Omron CX-Programmer project WWFH320 (CX-Programmer 9.73)

# PLC CPM2A: CPM2* 

## Global symbols (name address type ; comment)
0.00 BOOL  ; $?St$Bk?_#[4] / LS1 AREA SENSOR / $?St$Bk?_#[4]
0.01 BOOL  ; LS2 index origin
0.02 BOOL  ; LS3A WORK DETECT
0.03 BOOL  ; LS3B WORK DETECT
0.04 BOOL  ; LS4A WORK DETECT
0.05 BOOL  ; LS4B WORK DETECT
0.06 BOOL  ; LS5A WORK DETECT
0.07 BOOL  ; LS5B WORK DETECT
0.08 BOOL  ; LS6A WORK DETECT
0.09 BOOL  ; LS6B WORK DETECT
10.00 BOOL  ; SSR1 index start
10.01 BOOL  ; $?St$Bk?_#[5] / SSR2 INDEX CW / �$?St$Bk?_#[5]
10.02 BOOL  ; $?St$Bk?_#[6] / SSR3 INDEX CCW / $?St$Bk?_#[6]
10.03 BOOL  ; SSR4 OK SIGNAL T
10.04 BOOL  ; SOL1 ROTALY TABL
10.05 BOOL  ; shower flow on
10.06 BOOL  ; SOL3 air blow on
11.01 BOOL  ; M2,M4 ON
11.02 BOOL  ; MS5 work rotatio
11.06 BOOL  ; PL5A CYCLE RUN(G
11.07 BOOL  ; PL5B CYCLE RUN(R
12 CHANNEL  ; 7seg out channel
12.04 BOOL  ; 7SEG BLANK
12.05 BOOL  ; PL3 HOME POSITIO
12.06 BOOL  ; $?St$Bk?_#[7] / PL4 ALARM / 堎忢$?St$Bk?_#[7]
12.07 BOOL  ; $?St$Bk?_#[8] / PUMP MOTOR ON / �$?St$Bk?_#[8]
18.00 BOOL  ; cycle time displ
18.01 BOOL  ; cycle time displ
18.02 BOOL  ; cycle time displ
1.00 BOOL  ; PS1 AIR PRESSURE
1.01 BOOL  ; $?St$Bk?_#[9] / WORK OK SIGNAL / $?St$Bk?_#[9]
1.02 BOOL  ; MS0 CONTROL POWE
1.03 BOOL  ; CP1 INDEX PROTEC
1.06 BOOL  ; TS1 CYCLE START
1.07 BOOL  ; PB5 2HAND丂INTER
1.08 BOOL  ; PB8 PUMP MOTOR O
1.09 BOOL  ; PB9 PUMP MOTOR O
1.10 BOOL  ; PB3 ORIGIN丂CHEC
1.11 BOOL  ; $?St$Bk?_#[10] / PB4 alarm reset / $?St$Bk?_#[10]
200.00 BOOL  ; $?St$Bk?_#[11] / WORK OK / 馨窸K$?St$Bk?_#[11]
20.00 BOOL  ; $?St$Bk?_#[12] / CYCLE HAND ON / �$?St$Bk?_#[12]
20.01 BOOL  ; $?St$Bk?_#[13] / CYCLE HAND OFF / $?St$Bk?_#[13]
20.02 BOOL  ; $?St$Bk?_#[14] / INDEX RIGHT / 草�$?St$Bk?_#[14]
20.04 BOOL  ; $?St$Bk?_#[15] / INDEX LEFT / 草棉$?St$Bk?_#[15]
20.06 BOOL  ; WORK ROTATION ON
20.07 BOOL  ; WORK ROTATION OF
20.08 BOOL  ; ROTALT TABLE DOW
20.09 BOOL  ; $?St$Bk?_#[16] / rotary table up / $?St$Bk?_#[16]
20.10 BOOL  ; $?St$Bk?_#[17] / SHOWER ON / 愻忩$?St$Bk?_#[17]
20.11 BOOL  ; $?St$Bk?_#[18] / SHOWER OFF / 愻忩$?St$Bk?_#[18]
20.12 BOOL  ; $?St$Bk?_#[19] / AIR BLOW ON / 幢�$?St$Bk?_#[19]
20.13 BOOL  ; $?St$Bk?_#[20] / AIR BLOW OFF / 幢$?St$Bk?_#[20]
210.00 BOOL  ; $?St$Bk?_#[21] / ALARM CODE SET / $?St$Bk?_#[21]
211.14 BOOL  ; ALARM CODE SHIFT
212.00 BOOL  ; $?St$Bk?_#[22] / ALARM CODE ON / �$?St$Bk?_#[22]
212.01 BOOL  ; $?St$Bk?_#[23] / NEXT NG CODE / 師$?St$Bk?_#[23]
212.02 BOOL  ; NEXT ALARM CODE
212.04 BOOL  ; ALARM CODE CLEAR
213.01 BOOL  ; $?St$Bk?_#[25] / ALARM CODE "B" / $?St$Bk?_#[25]
213.02 BOOL  ; $?St$Bk?_#[26] / ALARM CODE "C" / $?St$Bk?_#[26]
213.03 BOOL  ; $?St$Bk?_#[27] / ALARM CODE "D" / $?St$Bk?_#[27]
220.00 BOOL  ; $?St$Bk?_#[28] / ALARM CODE OFF / $?St$Bk?_#[28]
23.00 BOOL  ; CONTROL POWER ON
23.01 BOOL  ; TS1 CYCLE START
23.02 BOOL  ; $?St$Bk?_#[29] / ORIGIN CHECK / 尨$?St$Bk?_#[29]
23.03 BOOL  ; $?St$Bk?_#[30] / ALARM RESET / 堎$?St$Bk?_#[30]
24.00 BOOL  ; $?St$Bk?_#[31] / INDEX ENABLE / 草$?St$Bk?_#[31]
253.08 BOOL  ; CPU BATTERY DOWN
253.10 BOOL  ; CPU I/O UNIT ERR
25.00 BOOL  ; HAND MODE丂INABL
26.00 BOOL  ; $?St$Bk?_#[32] / INDEX RIGHT / 草�$?St$Bk?_#[32]
26.02 BOOL  ; $?St$Bk?_#[33] / INDEX LEFT / 草棉$?St$Bk?_#[33]
26.04 BOOL  ; $?St$Bk?_#[34] / INDEX RIGHT / 草�$?St$Bk?_#[34]
26.06 BOOL  ; $?St$Bk?_#[35] / INDEX RIGHT / 草�$?St$Bk?_#[35]
26.08 BOOL  ; $?St$Bk?_#[36] / INDEX RIGHT END / $?St$Bk?_#[36]
26.10 BOOL  ; $?St$Bk?_#[37] / INDEX LEFT / 草棉$?St$Bk?_#[37]
26.12 BOOL  ; $?St$Bk?_#[38] / INDEX LEFT / 草棉$?St$Bk?_#[38]
26.14 BOOL  ; $?St$Bk?_#[39] / INDEX LEFT END / $?St$Bk?_#[39]
27.00 BOOL  ; WORK ROTATION ON
27.02 BOOL  ; WORK ROTATION OF
27.06 BOOL  ; $?St$Bk?_#[40] / SHOWER ON / 愻忩$?St$Bk?_#[40]
27.08 BOOL  ; $?St$Bk?_#[41] / SHOWER OFF / 愻忩$?St$Bk?_#[41]
27.10 BOOL  ; $?St$Bk?_#[42] / SHOWER ON / 愻忩$?St$Bk?_#[42]
27.12 BOOL  ; rotary table dow
27.14 BOOL  ; $?St$Bk?_#[43] / rotary table up / $?St$Bk?_#[43]
28.00 BOOL  ; $?St$Bk?_#[44] / AIR BLOW ON / 幢�$?St$Bk?_#[44]
28.02 BOOL  ; $?St$Bk?_#[45] / AIR BLOW OFF / 幢$?St$Bk?_#[45]
29.00 BOOL  ; $?St$Bk?_#[46] / PUMP MOTOR ON / �$?St$Bk?_#[46]
2.00 BOOL  ; $?St$Bk?_#[47] / SS1 CYCLE HAND / $?St$Bk?_#[47]
2.01 BOOL  ; $?St$Bk?_#[48] / SS2 INDEX RIGHT / $?St$Bk?_#[48]
2.02 BOOL  ; $?St$Bk?_#[49] / SS2 INDEX LEFT / $?St$Bk?_#[49]
2.03 BOOL  ; SS3 WORK ROTATIO
2.04 BOOL  ; SS4 ROTALT TABLE
2.05 BOOL  ; $?St$Bk?_#[50] / SS5 SHOWER ON / $?St$Bk?_#[50]
2.06 BOOL  ; $?St$Bk?_#[51] / SS6 AIR BLOW ON / $?St$Bk?_#[51]
2.07 BOOL  ; SW1 WORK DETECT
2.08 BOOL  ; WASHER FLOW SWIT
2.10 BOOL  ; FS2 WASHER LIQUI
30.00 BOOL  ; return cycle run
30.01 BOOL  ; return cycle 1cm
30.02 BOOL  ; return cycle 2cm
30.13 BOOL  ; return cycle ind
30.14 BOOL  ; return cycle ind
30.15 BOOL  ; return complete
31.00 BOOL  ; WORK DETECT IN 1
31.01 BOOL  ; WORK DETECT IN 2
31.02 BOOL  ; NO WORK DETECT I
31.03 BOOL  ; $?St$Bk?_#[52] / WORK DETECT OUT / $?St$Bk?_#[52]
31.04 BOOL  ; NO WORK DETECT O
31.05 BOOL  ; WORK DETECT IN丂
31.06 BOOL  ; WORK DETECT IN俀
32.00 BOOL  ; $?St$Bk?_#[53] / HAND MODE / 庤摦�$?St$Bk?_#[53]
32.01 BOOL  ; $?St$Bk?_#[54] / CYCLE AUTO / 帺摦$?St$Bk?_#[54]
32.05 BOOL  ; work OK signal c
32.09 BOOL  ; $?St$Bk?_#[55] / MAIN AIR OK / 嬻$?St$Bk?_#[55]
32.10 BOOL  ; $?St$Bk?_#[56] / SWITCH OK / AUTO$?St$Bk?_#[56]
32.11 BOOL  ; $?St$Bk?_#[57] / SWITCH OK / 讲�罯$?St$Bk?_#[57]
32.12 BOOL  ; $?St$Bk?_#[58] / LS OK / 匦�慕帛罯$?St$Bk?_#[58]
32.13 BOOL  ; $?St$Bk?_#[59] / SOL OK / 口刹霓OK$?St$Bk?_#[59]
32.14 BOOL  ; INDEX PROTECTOR
32.15 BOOL  ; $?St$Bk?_#[60] / MACHIN ORIGIN / $?St$Bk?_#[60]
33.00 BOOL  ; $?St$Bk?_#[61] / EMERGENCY STOP / $?St$Bk?_#[61]
33.02 BOOL  ; $?St$Bk?_#[62] / CYCLE STOP / 徊纲$?St$Bk?_#[62]
33.15 BOOL  ; $?St$Bk?_#[63] / HOME POSITION / $?St$Bk?_#[63]
34.00 BOOL  ; $?St$Bk?_#[64] / CYCLE RUN / 婲摦$?St$Bk?_#[64]
34.01 BOOL  ; $?St$Bk?_#[65] / CYCLE START / 徊�$?St$Bk?_#[65]
34.02 BOOL  ; cycle stat comma
34.03 BOOL  ; CYCLE MEMORY CLE
34.04 BOOL  ; work=1丄馨�1屄棳
34.05 BOOL  ; 楢懕徊纲
34.06 BOOL  ; $?St$Bk?_#[66] / AUTO CYCLE OFF / $?St$Bk?_#[66]
3.00 BOOL  ; LS7 rotary table
3.01 BOOL  ; LS8 ROTARY TABLE
3.02 BOOL  ; THR1 CLEAN TANK
3.06 BOOL  ; OL2 WASHER PUMP
3.08 BOOL  ; OL4 MISTPURE MOT
3.09 BOOL  ; OL5 WORK ROTATIO
3.10 BOOL  ; M2 M4 ON
40.00 BOOL  ; index right comm
40.02 BOOL  ; index right turn
40.04 BOOL  ; iindex right fin
40.06 BOOL  ; rotary table not
41.00 BOOL  ; rotary table dow
41.01 BOOL  ; rotary table dow
41.02 BOOL  ; work rotation mo
41.03 BOOL  ; $?St$Bk?_#[67] / shower flow fin / $?St$Bk?_#[67]
41.04 BOOL  ; air brow command
41.05 BOOL  ; $?St$Bk?_#[68] / air brow fin / 幢$?St$Bk?_#[68]
41.06 BOOL  ; work丂rotaition
41.07 BOOL  ; work丂rotaition
41.08 BOOL  ; rotary table up
41.09 BOOL  ; rotary table up
42.00 BOOL  ; $?St$Bk?_#[69] / first cycle end / $?St$Bk?_#[69]
42.01 BOOL  ; $?St$Bk?_#[70] / 2nd cycle end / $?St$Bk?_#[70]
42.02 BOOL  ; 2nd cycle start
42.04 BOOL  ; $?St$Bk?_#[71] / 2nd cycle end / $?St$Bk?_#[71]
47.00 BOOL  ; $?St$Bk?_#[72] / index right / 草�$?St$Bk?_#[72]
47.02 BOOL  ; index right turn
47.04 BOOL  ; $?St$Bk?_#[73] / index right end / $?St$Bk?_#[73]
49.00 BOOL  ; $?St$Bk?_#[74] / cycle Ffinish / $?St$Bk?_#[74]
DM0 CHANNEL  ; PROGRAM VERSION
DM1 CHANNEL  ; CYCLE TIME COUNT
DM10 CHANNEL  ; $?St$Bk?_#[75] / CYCLE COUNT / 徊�$?St$Bk?_#[75]
DM120 CHANNEL  ; shower flow time
DM121 CHANNEL  ; $?St$Bk?_#[76] / air blow timer / $?St$Bk?_#[76]
DM2 CHANNEL  ; CYCLE TIME
HR10.00 BOOL  ; AIR PRESSURE ALA
HR10.02 BOOL  ; WASHER PUMP MOTO
HR10.03 BOOL  ; 丂
HR10.04 BOOL  ; MISTPURE MOTOR O
HR10.05 BOOL  ; WORK ROTATION  M
HR10.06 BOOL  ; $?St$Bk?_#[77] / AREA SENSOR OFF / $?St$Bk?_#[77]
HR10.07 BOOL  ; NDEX PROTECTOR N
HR10.08 BOOL  ; CONTROL POWER OF
HR10.09 BOOL  ; $?St$Bk?_#[78] / PLC丂ALARM / 及馆$?St$Bk?_#[78]
HR11.00 BOOL  ; INDEX TIME OVER
HR11.01 BOOL  ; ROTALY TABLE UP/
HR11.03 BOOL  ; M2,M4 ALARM
HR11.04 BOOL  ; WASHER FLOW SWIT
HR11.08 BOOL  ; $?St$Bk?_#[79] / INDEX WORK NG / �$?St$Bk?_#[79]
HR11.09 BOOL  ; $?St$Bk?_#[80] / CYCLE TIME OVER / $?St$Bk?_#[80]
HR11.15 BOOL  ; return cycle tim
HR12.00 BOOL  ; $?St$Bk?_#[81] / LS POSITION NG / $?St$Bk?_#[81]
HR12.01 BOOL  ; SWITCH POSITION
HR12.02 BOOL  ; IOK SIGNAL NOT C
HR12.04 BOOL  ; WORK DETECT IN N
HR12.05 BOOL  ; WORK DETECT OUT
HR12.06 BOOL  ; $?St$Bk?_#[82] / SOL NG / 口刹霓尨$?St$Bk?_#[82]
HR13.00 BOOL  ; SWITCH POSITION
HR13.02 BOOL  ; CLEAN TANK TEMP
HR13.03 BOOL  ; $?St$Bk?_#[83] / WASHER LEVEL NG / $?St$Bk?_#[83]
HR14.00 BOOL  ; EMERGENCY STOP A
HR14.01 BOOL  ; EMERGENCY STOP A
HR14.02 BOOL  ; EMERGENCY STOP A
HR14.03 BOOL  ; CYCLE STOP ALARM
HR14.10 BOOL  ; $?St$Bk?_#[84] / ALARM / 憤崌堎忢$?St$Bk?_#[84]
HR14.11 BOOL  ; $?St$Bk?_#[85] / ALARM ON / 弊把敪$?St$Bk?_#[85]
HR19.00 BOOL  ; 嫙媼晹馨妇莼皸L
TIM000 BOOL  ; CYCLE TIME OVER
TIM002 BOOL  ; 2HAND INTERLOCK
TIM005 BOOL  ; $?St$Bk?_#[86] / alarm reset ON / $?St$Bk?_#[86]
TIM009 BOOL  ; rotary table dow
TIM010 BOOL  ; $?St$Bk?_#[87] / INDEX RIGTH END / $?St$Bk?_#[87]
TIM011 BOOL  ; shower flow time
TIM012 BOOL  ; $?St$Bk?_#[88] / air blow timer / $?St$Bk?_#[88]
TIM013 BOOL  ; work丂rotation m
TIM020 BOOL  ; INDEX TIME OVER
TIM021 BOOL  ; ROTALY TABLE UP/
TIM023 BOOL  ; M2,M4 ALARM
TIM025 BOOL  ; WASHER FLOW SWIT
TIM029 BOOL  ; 楢懕徊纲婲摦
TIM030 BOOL  ; SOL2 shower flow
TIM031 BOOL  ; SOL2 shower flow
TIM050 BOOL  ; ALARM CODE A TO
TIM051 BOOL  ; ALARM CODE 0 TO
TIM052 BOOL  ; NEXT ALARM CODE
TIM130 BOOL  ; return start che
TIM131 BOOL  ; return cycle tim
TIM133 BOOL  ; return cycle com

## Program 怴婯踢鄹拮�1 (no task)

### Section VERSION
; 这套PLC程序设计用于控制一台轴承自动检测机，与上位机NT31-ST123协同工作。 / 程序实现了手动和自动两种操作模式。 / 将PLC控制器，连接循环手动开关、索引开关、工件旋转开关、旋转台开关、喷淋开关、气吹开关、双手互锁按钮、工件检测传感器、原点位置传感器、气压检测传感器、清洗泵、气吹装置、报警灯、7段显示器等设备。 / 在手动模式下，操作员通过按下循环手动开关切换模式，置位手动模式使能，即可通过索引右开关和索引左开关控制索引启动继电器的方向，调整轴承位置。按下工件旋转开关触发工件旋转电机控制继电器，使工件旋转以便检查。通过旋转台开关操作旋转台控制电磁阀升降旋转台，但下降时需双手互锁开关置位以保障安全。按下喷淋开关开启喷淋控制电磁阀进行清洗，或按下气吹开关启动气吹控制电磁阀吹干水分。手动操作通过7段显示输出通道实时展示状态。 / 在自动模式下，操作员按下循环启动按钮触发流程，系统检查原点位置标志是否置位，只有设备处于原点位置时循环运行标志才会置位并开始运行，同时需确保工件检测传感器A和工件检测传感器B置位以确认工件到位。若双手互锁置位且循环启动触发，系统进入自动模式准备状态。当循环启动命令置位后，系统记录工件检测状态以备后续检查。若工件检测B与开关同时置位，确认工件到位信号。自动流程按顺序执行：索引启动继电器将轴承移至检测位，旋转台控制电磁阀下降至清洗位，工件旋转电机控制继电器启动以均匀清洗轴承表面。接着，喷淋控制电磁阀开启进行清洗，此时需工件检测传感器A置位以确认工件存在。随后，气吹控制电磁阀吹干水分，需旋转台下降传感器置位以保证旋转台在下降位。当旋转台下降传感器置位时，确认旋转台下降到位信号。清洗吹干完成后，旋转台控制电磁阀上升复位，循环计数存储记录检测次数，最终通过OK信号继电器输出检测结果。 / 运行过程中，系统通过7段显示输出通道显示状态。若气压检测传感器检测到气压低于阈值或清洗泵过载传感器置位，循环运行标志立即复位，报警指示灯亮起，7段显示输出通道显示报警代码，系统进入紧急停止标志状态。操作员按下报警复位按钮后，只有当所有异常条件清除时，报警指示灯才会熄灭，系统恢复运行。

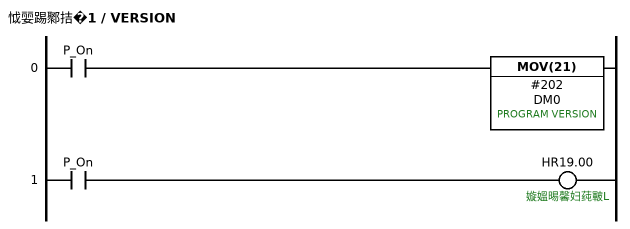
; rung 0
LD P_On
MOV(21) #202 DM0  ; PROGRAM VERSION
; rung 1
LD P_On
OUT HR19.00  ; 嫙媼晹馨妇莼皸L

### Section CYCLE_SET

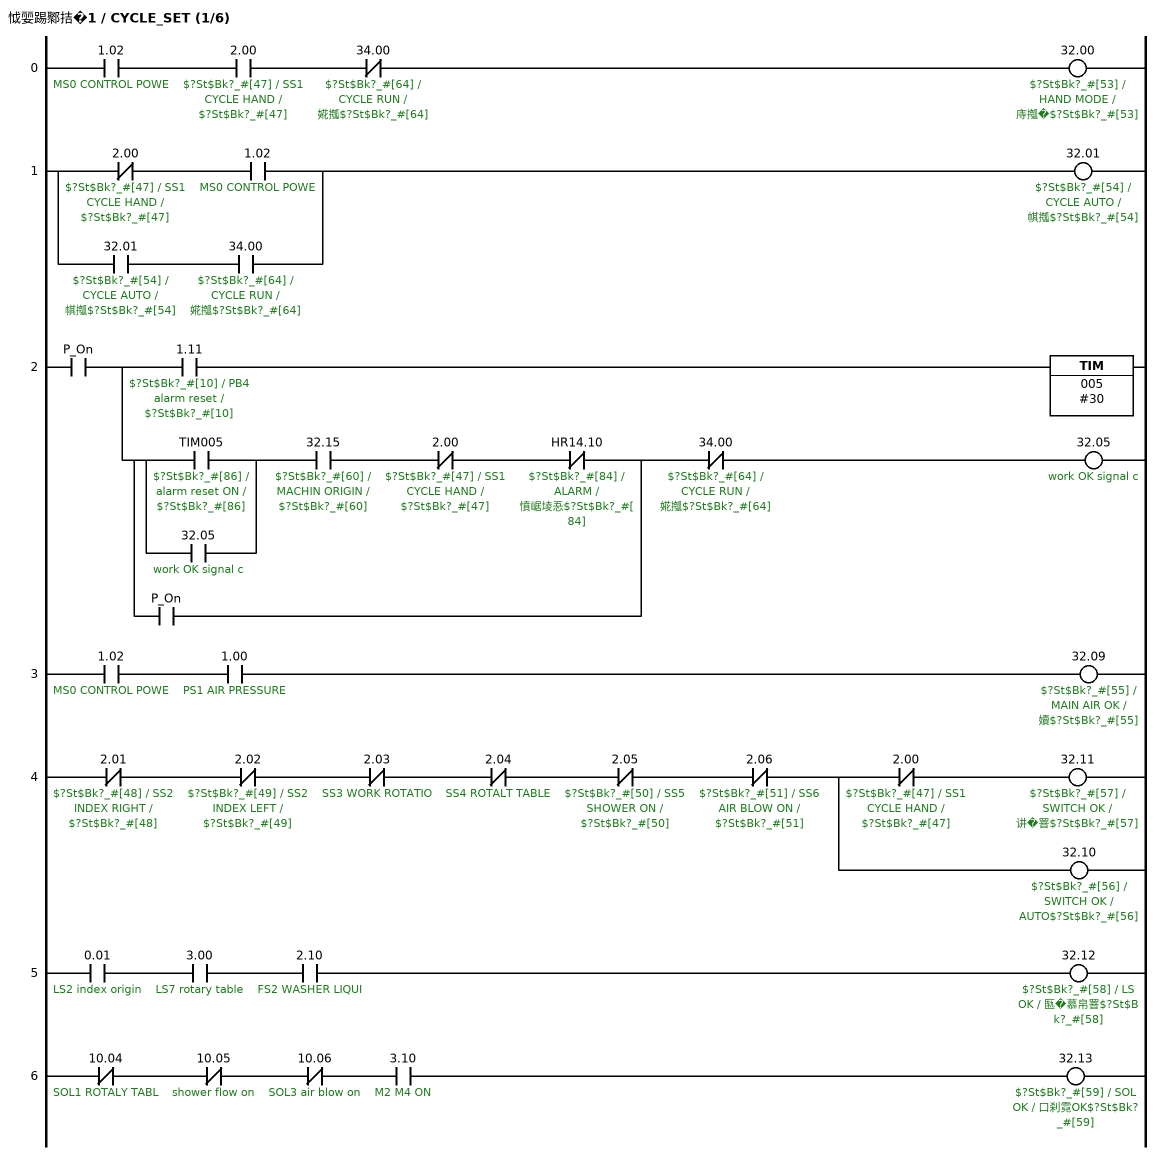
; rung 0
LD 1.02  ; MS0 CONTROL POWE
AND 2.00  ; $?St$Bk?_#[47] / SS1 CYCLE HAND / $?St$Bk?_#[47]
ANDNOT 34.00  ; $?St$Bk?_#[64] / CYCLE RUN / 婲摦$?St$Bk?_#[64]
OUT 32.00  ; $?St$Bk?_#[53] / HAND MODE / 庤摦�$?St$Bk?_#[53]
; rung 1
LDNOT 2.00  ; $?St$Bk?_#[47] / SS1 CYCLE HAND / $?St$Bk?_#[47]
AND 1.02  ; MS0 CONTROL POWE
LD 32.01  ; $?St$Bk?_#[54] / CYCLE AUTO / 帺摦$?St$Bk?_#[54]
AND 34.00  ; $?St$Bk?_#[64] / CYCLE RUN / 婲摦$?St$Bk?_#[64]
ORLD
OUT 32.01  ; $?St$Bk?_#[54] / CYCLE AUTO / 帺摦$?St$Bk?_#[54]
; rung 2
LD P_On
OUT TR0
AND 1.11  ; $?St$Bk?_#[10] / PB4 alarm reset / $?St$Bk?_#[10]
TIM 005 #30
LD TR0
LD TIM005  ; $?St$Bk?_#[86] / alarm reset ON / $?St$Bk?_#[86]
OR 32.05  ; work OK signal c
AND 32.15  ; $?St$Bk?_#[60] / MACHIN ORIGIN / $?St$Bk?_#[60]
ANDNOT 2.00  ; $?St$Bk?_#[47] / SS1 CYCLE HAND / $?St$Bk?_#[47]
ANDNOT HR14.10  ; $?St$Bk?_#[84] / ALARM / 憤崌堎忢$?St$Bk?_#[84]
OR P_On
ANDLD
ANDNOT 34.00  ; $?St$Bk?_#[64] / CYCLE RUN / 婲摦$?St$Bk?_#[64]
OUT 32.05  ; work OK signal c
; rung 3
LD 1.02  ; MS0 CONTROL POWE
AND 1.00  ; PS1 AIR PRESSURE
OUT 32.09  ; $?St$Bk?_#[55] / MAIN AIR OK / 嬻$?St$Bk?_#[55]
; rung 4
LDNOT 2.01  ; $?St$Bk?_#[48] / SS2 INDEX RIGHT / $?St$Bk?_#[48]
ANDNOT 2.02  ; $?St$Bk?_#[49] / SS2 INDEX LEFT / $?St$Bk?_#[49]
ANDNOT 2.03  ; SS3 WORK ROTATIO
ANDNOT 2.04  ; SS4 ROTALT TABLE
ANDNOT 2.05  ; $?St$Bk?_#[50] / SS5 SHOWER ON / $?St$Bk?_#[50]
ANDNOT 2.06  ; $?St$Bk?_#[51] / SS6 AIR BLOW ON / $?St$Bk?_#[51]
OUT TR0
ANDNOT 2.00  ; $?St$Bk?_#[47] / SS1 CYCLE HAND / $?St$Bk?_#[47]
OUT 32.11  ; $?St$Bk?_#[57] / SWITCH OK / 讲�罯$?St$Bk?_#[57]
LD TR0
OUT 32.10  ; $?St$Bk?_#[56] / SWITCH OK / AUTO$?St$Bk?_#[56]
; rung 5
LD 0.01  ; LS2 index origin
AND 3.00  ; LS7 rotary table
AND 2.10  ; FS2 WASHER LIQUI
OUT 32.12  ; $?St$Bk?_#[58] / LS OK / 匦�慕帛罯$?St$Bk?_#[58]
; rung 6
LDNOT 10.04  ; SOL1 ROTALY TABL
ANDNOT 10.05  ; shower flow on
ANDNOT 10.06  ; SOL3 air blow on
AND 3.10  ; M2 M4 ON
OUT 32.13  ; $?St$Bk?_#[59] / SOL OK / 口刹霓OK$?St$Bk?_#[59]

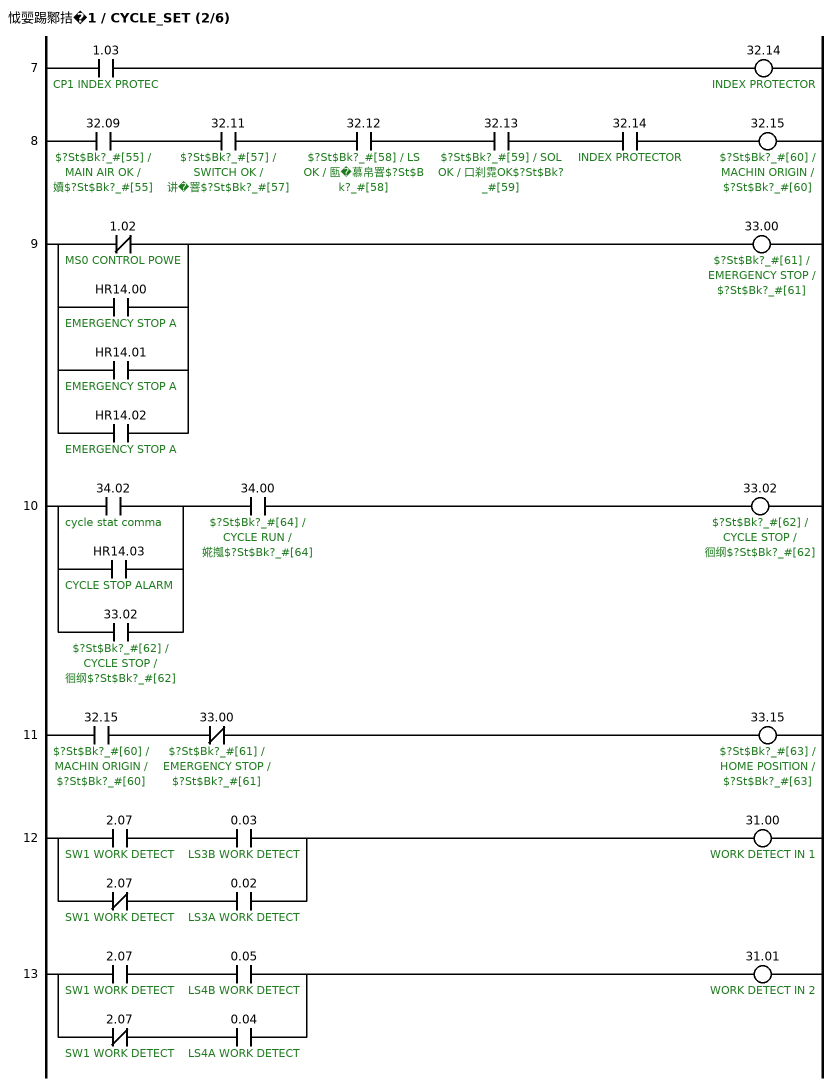
; rung 7
LD 1.03  ; CP1 INDEX PROTEC
OUT 32.14  ; INDEX PROTECTOR
; rung 8
LD 32.09  ; $?St$Bk?_#[55] / MAIN AIR OK / 嬻$?St$Bk?_#[55]
AND 32.11  ; $?St$Bk?_#[57] / SWITCH OK / 讲�罯$?St$Bk?_#[57]
AND 32.12  ; $?St$Bk?_#[58] / LS OK / 匦�慕帛罯$?St$Bk?_#[58]
AND 32.13  ; $?St$Bk?_#[59] / SOL OK / 口刹霓OK$?St$Bk?_#[59]
AND 32.14  ; INDEX PROTECTOR
OUT 32.15  ; $?St$Bk?_#[60] / MACHIN ORIGIN / $?St$Bk?_#[60]
; rung 9
LDNOT 1.02  ; MS0 CONTROL POWE
OR HR14.00  ; EMERGENCY STOP A
OR HR14.01  ; EMERGENCY STOP A
OR HR14.02  ; EMERGENCY STOP A
OUT 33.00  ; $?St$Bk?_#[61] / EMERGENCY STOP / $?St$Bk?_#[61]
; rung 10
LD 34.02  ; cycle stat comma
OR HR14.03  ; CYCLE STOP ALARM
OR 33.02  ; $?St$Bk?_#[62] / CYCLE STOP / 徊纲$?St$Bk?_#[62]
AND 34.00  ; $?St$Bk?_#[64] / CYCLE RUN / 婲摦$?St$Bk?_#[64]
OUT 33.02  ; $?St$Bk?_#[62] / CYCLE STOP / 徊纲$?St$Bk?_#[62]
; rung 11
LD 32.15  ; $?St$Bk?_#[60] / MACHIN ORIGIN / $?St$Bk?_#[60]
ANDNOT 33.00  ; $?St$Bk?_#[61] / EMERGENCY STOP / $?St$Bk?_#[61]
OUT 33.15  ; $?St$Bk?_#[63] / HOME POSITION / $?St$Bk?_#[63]
; rung 12
LD 2.07  ; SW1 WORK DETECT
AND 0.03  ; LS3B WORK DETECT
LDNOT 2.07  ; SW1 WORK DETECT
AND 0.02  ; LS3A WORK DETECT
ORLD
OUT 31.00  ; WORK DETECT IN 1
; rung 13
LD 2.07  ; SW1 WORK DETECT
AND 0.05  ; LS4B WORK DETECT
LDNOT 2.07  ; SW1 WORK DETECT
AND 0.04  ; LS4A WORK DETECT
ORLD
OUT 31.01  ; WORK DETECT IN 2

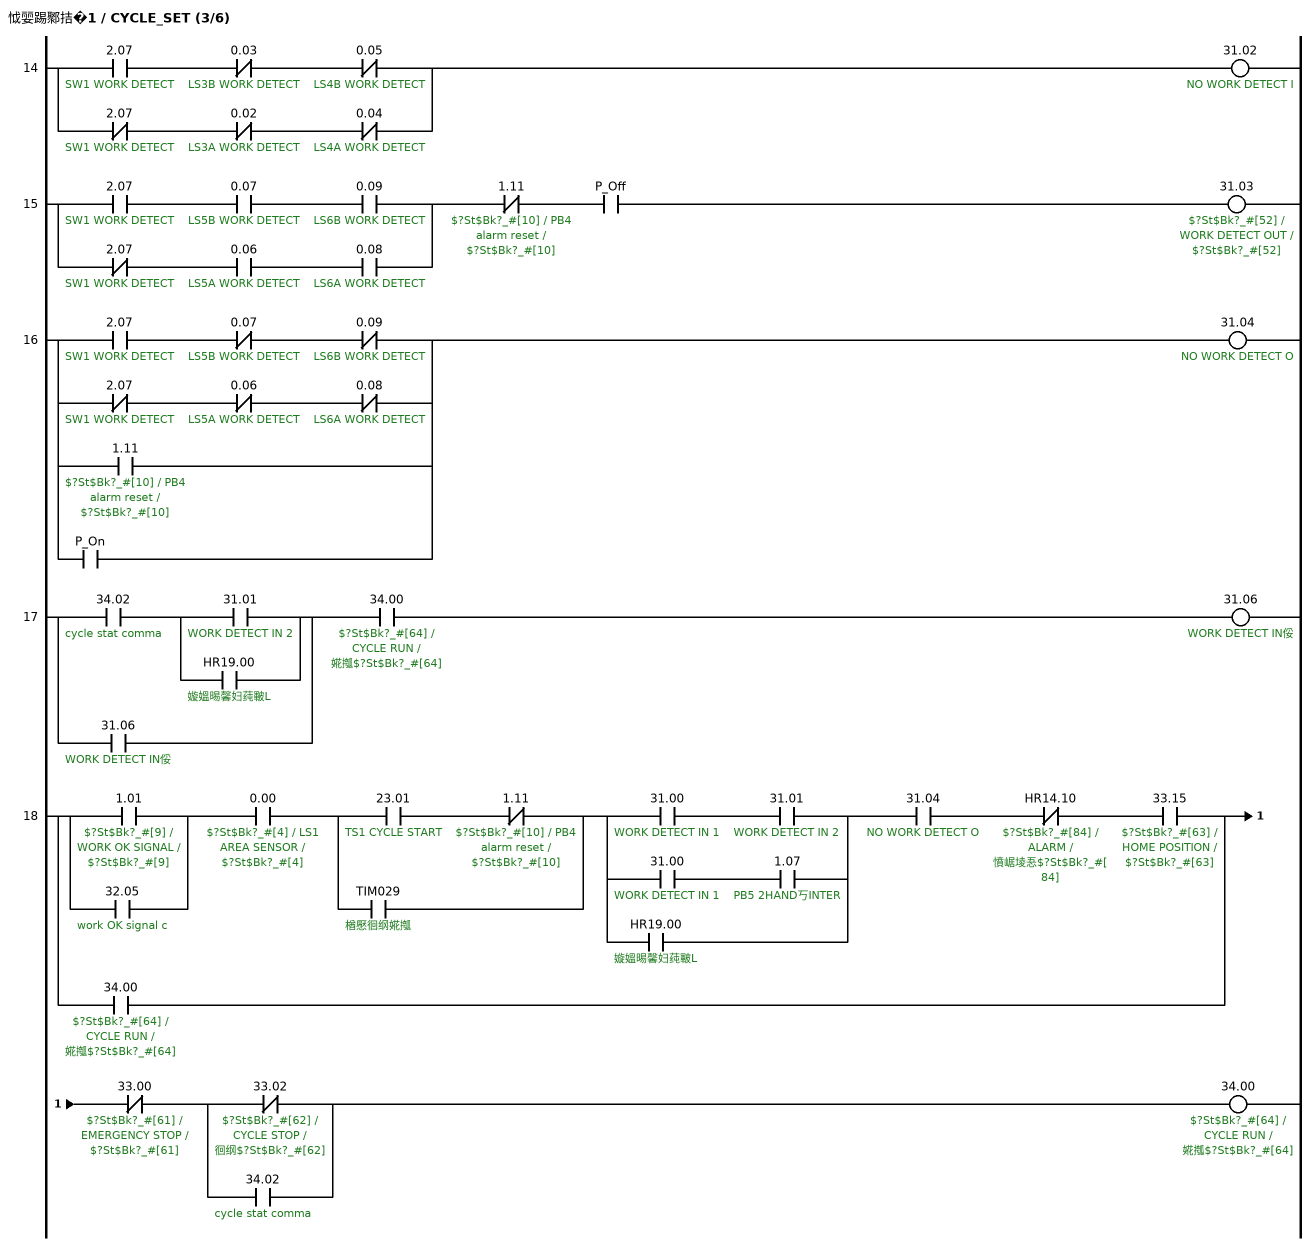
; rung 14
LD 2.07  ; SW1 WORK DETECT
ANDNOT 0.03  ; LS3B WORK DETECT
ANDNOT 0.05  ; LS4B WORK DETECT
LDNOT 2.07  ; SW1 WORK DETECT
ANDNOT 0.02  ; LS3A WORK DETECT
ANDNOT 0.04  ; LS4A WORK DETECT
ORLD
OUT 31.02  ; NO WORK DETECT I
; rung 15
LD 2.07  ; SW1 WORK DETECT
AND 0.07  ; LS5B WORK DETECT
AND 0.09  ; LS6B WORK DETECT
LDNOT 2.07  ; SW1 WORK DETECT
AND 0.06  ; LS5A WORK DETECT
AND 0.08  ; LS6A WORK DETECT
ORLD
ANDNOT 1.11  ; $?St$Bk?_#[10] / PB4 alarm reset / $?St$Bk?_#[10]
AND P_Off
OUT 31.03  ; $?St$Bk?_#[52] / WORK DETECT OUT / $?St$Bk?_#[52]
; rung 16
LD 2.07  ; SW1 WORK DETECT
ANDNOT 0.07  ; LS5B WORK DETECT
ANDNOT 0.09  ; LS6B WORK DETECT
LDNOT 2.07  ; SW1 WORK DETECT
ANDNOT 0.06  ; LS5A WORK DETECT
ANDNOT 0.08  ; LS6A WORK DETECT
ORLD
LD 1.11  ; $?St$Bk?_#[10] / PB4 alarm reset / $?St$Bk?_#[10]
OR P_On
ORLD
OUT 31.04  ; NO WORK DETECT O
; rung 17
LD 34.02  ; cycle stat comma
LD 31.01  ; WORK DETECT IN 2
OR HR19.00  ; 嫙媼晹馨妇莼皸L
ANDLD
OR 31.06  ; WORK DETECT IN俀
AND 34.00  ; $?St$Bk?_#[64] / CYCLE RUN / 婲摦$?St$Bk?_#[64]
OUT 31.06  ; WORK DETECT IN俀
; rung 18
LD 1.01  ; $?St$Bk?_#[9] / WORK OK SIGNAL / $?St$Bk?_#[9]
OR 32.05  ; work OK signal c
AND 0.00  ; $?St$Bk?_#[4] / LS1 AREA SENSOR / $?St$Bk?_#[4]
LD 23.01  ; TS1 CYCLE START
ANDNOT 1.11  ; $?St$Bk?_#[10] / PB4 alarm reset / $?St$Bk?_#[10]
OR TIM029  ; 楢懕徊纲婲摦
ANDLD
LD 31.00  ; WORK DETECT IN 1
AND 31.01  ; WORK DETECT IN 2
LD 31.00  ; WORK DETECT IN 1
AND 1.07  ; PB5 2HAND丂INTER
ORLD
OR HR19.00  ; 嫙媼晹馨妇莼皸L
ANDLD
AND 31.04  ; NO WORK DETECT O
ANDNOT HR14.10  ; $?St$Bk?_#[84] / ALARM / 憤崌堎忢$?St$Bk?_#[84]
AND 33.15  ; $?St$Bk?_#[63] / HOME POSITION / $?St$Bk?_#[63]
OR 34.00  ; $?St$Bk?_#[64] / CYCLE RUN / 婲摦$?St$Bk?_#[64]
ANDNOT 33.00  ; $?St$Bk?_#[61] / EMERGENCY STOP / $?St$Bk?_#[61]
LDNOT 33.02  ; $?St$Bk?_#[62] / CYCLE STOP / 徊纲$?St$Bk?_#[62]
OR 34.02  ; cycle stat comma
ANDLD
OUT 34.00  ; $?St$Bk?_#[64] / CYCLE RUN / 婲摦$?St$Bk?_#[64]

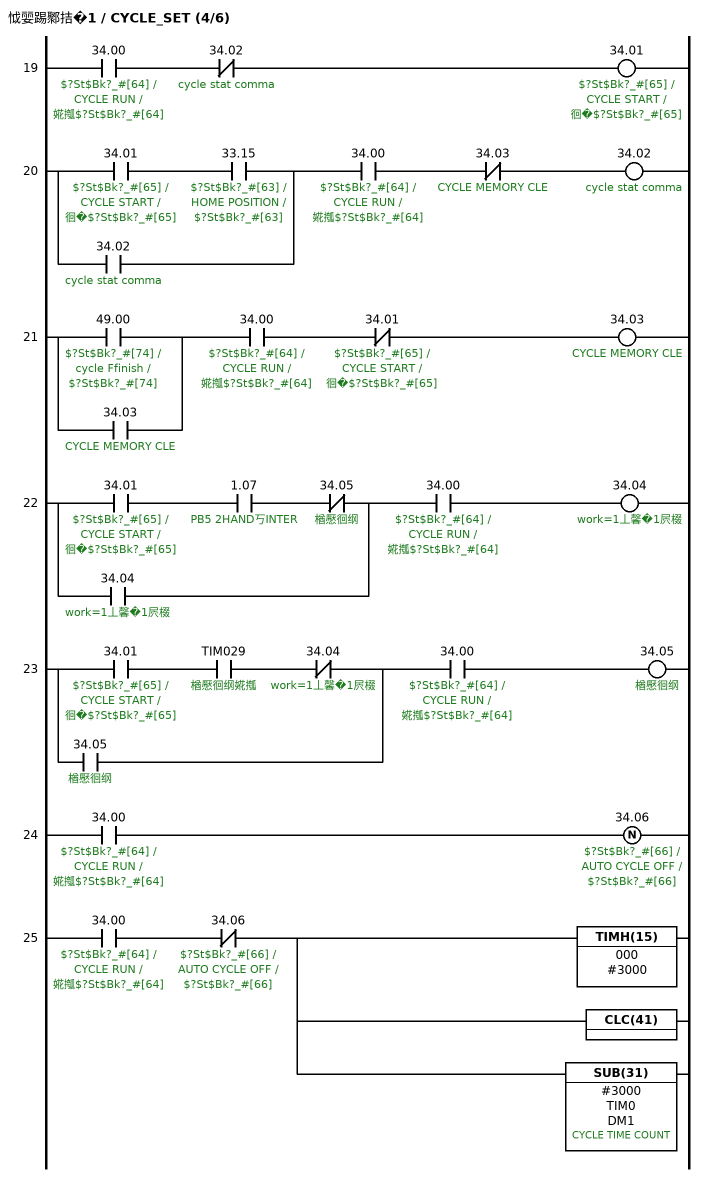
; rung 19
LD 34.00  ; $?St$Bk?_#[64] / CYCLE RUN / 婲摦$?St$Bk?_#[64]
ANDNOT 34.02  ; cycle stat comma
OUT 34.01  ; $?St$Bk?_#[65] / CYCLE START / 徊�$?St$Bk?_#[65]
; rung 20
LD 34.01  ; $?St$Bk?_#[65] / CYCLE START / 徊�$?St$Bk?_#[65]
AND 33.15  ; $?St$Bk?_#[63] / HOME POSITION / $?St$Bk?_#[63]
OR 34.02  ; cycle stat comma
AND 34.00  ; $?St$Bk?_#[64] / CYCLE RUN / 婲摦$?St$Bk?_#[64]
ANDNOT 34.03  ; CYCLE MEMORY CLE
OUT 34.02  ; cycle stat comma
; rung 21
LD 49.00  ; $?St$Bk?_#[74] / cycle Ffinish / $?St$Bk?_#[74]
OR 34.03  ; CYCLE MEMORY CLE
AND 34.00  ; $?St$Bk?_#[64] / CYCLE RUN / 婲摦$?St$Bk?_#[64]
ANDNOT 34.01  ; $?St$Bk?_#[65] / CYCLE START / 徊�$?St$Bk?_#[65]
OUT 34.03  ; CYCLE MEMORY CLE
; rung 22
LD 34.01  ; $?St$Bk?_#[65] / CYCLE START / 徊�$?St$Bk?_#[65]
AND 1.07  ; PB5 2HAND丂INTER
ANDNOT 34.05  ; 楢懕徊纲
OR 34.04  ; work=1丄馨�1屄棳
AND 34.00  ; $?St$Bk?_#[64] / CYCLE RUN / 婲摦$?St$Bk?_#[64]
OUT 34.04  ; work=1丄馨�1屄棳
; rung 23
LD 34.01  ; $?St$Bk?_#[65] / CYCLE START / 徊�$?St$Bk?_#[65]
AND TIM029  ; 楢懕徊纲婲摦
ANDNOT 34.04  ; work=1丄馨�1屄棳
OR 34.05  ; 楢懕徊纲
AND 34.00  ; $?St$Bk?_#[64] / CYCLE RUN / 婲摦$?St$Bk?_#[64]
OUT 34.05  ; 楢懕徊纲
; rung 24
LD 34.00  ; $?St$Bk?_#[64] / CYCLE RUN / 婲摦$?St$Bk?_#[64]
DIFD(14) 34.06  ; $?St$Bk?_#[66] / AUTO CYCLE OFF / $?St$Bk?_#[66]
; rung 25
LD 34.00  ; $?St$Bk?_#[64] / CYCLE RUN / 婲摦$?St$Bk?_#[64]
ANDNOT 34.06  ; $?St$Bk?_#[66] / AUTO CYCLE OFF / $?St$Bk?_#[66]
TIMH(15) 000 #3000
CLC(41)
SUB(31) #3000 TIM0 DM1  ; CYCLE TIME COUNT

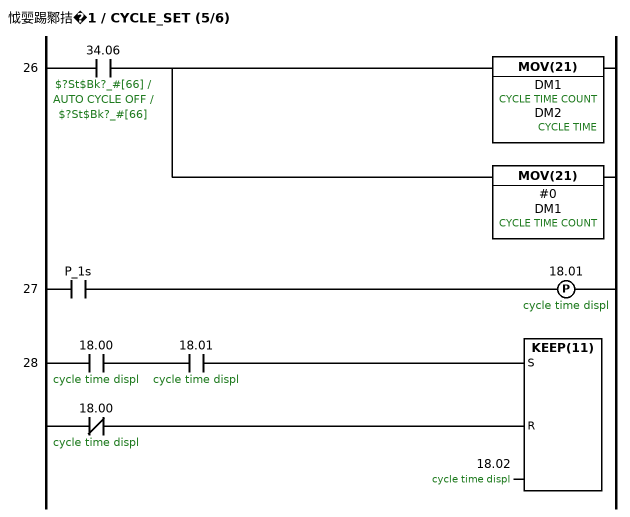
; rung 26
LD 34.06  ; $?St$Bk?_#[66] / AUTO CYCLE OFF / $?St$Bk?_#[66]
MOV(21) DM1 DM2  ; CYCLE TIME COUNT, CYCLE TIME
MOV(21) #0 DM1  ; CYCLE TIME COUNT
; rung 27
LD P_1s
DIFU(13) 18.01  ; cycle time displ
; rung 28
LD 18.00  ; cycle time displ
AND 18.01  ; cycle time displ
LDNOT 18.00  ; cycle time displ
KEEP(11) 18.02  ; cycle time displ

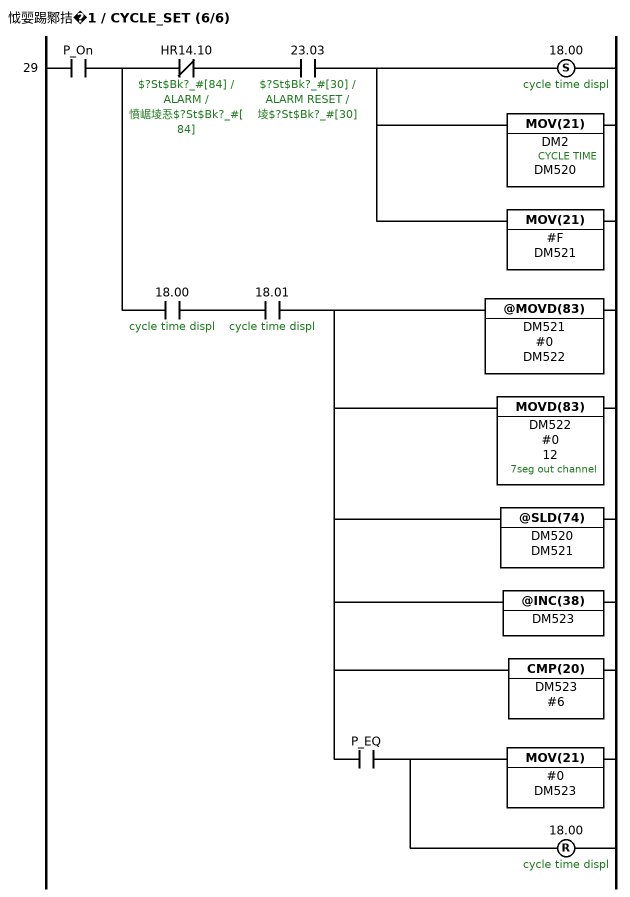
; rung 29
LD P_On
OUT TR0
ANDNOT HR14.10  ; $?St$Bk?_#[84] / ALARM / 憤崌堎忢$?St$Bk?_#[84]
AND 23.03  ; $?St$Bk?_#[30] / ALARM RESET / 堎$?St$Bk?_#[30]
SET 18.00  ; cycle time displ
MOV(21) DM2 DM520  ; CYCLE TIME
MOV(21) #F DM521
LD TR0
AND 18.00  ; cycle time displ
AND 18.01  ; cycle time displ
@MOVD(83) DM521 #0 DM522
MOVD(83) DM522 #0 12  ; 7seg out channel
@SLD(74) DM520 DM521
@INC(38) DM523
CMP(20) DM523 #6
AND P_EQ
MOV(21) #0 DM523
RSET 18.00  ; cycle time displ

### Section AUTO_CYCLE

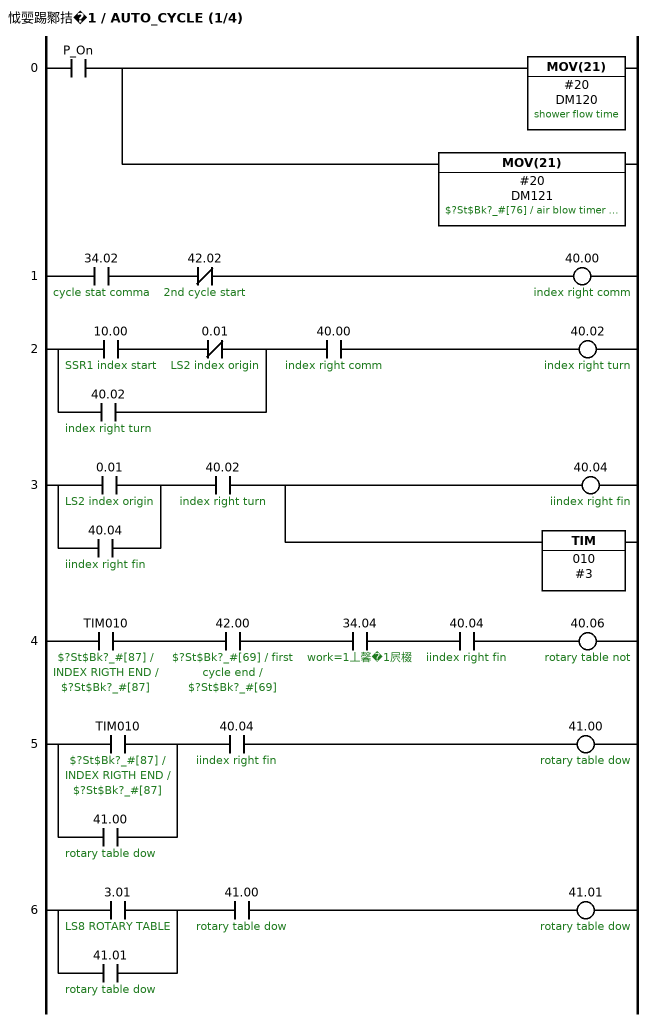
; rung 0
LD P_On
MOV(21) #20 DM120  ; shower flow time
MOV(21) #20 DM121  ; $?St$Bk?_#[76] / air blow timer / $?St$Bk?_#[76]
; rung 1
LD 34.02  ; cycle stat comma
ANDNOT 42.02  ; 2nd cycle start
OUT 40.00  ; index right comm
; rung 2
LD 10.00  ; SSR1 index start
ANDNOT 0.01  ; LS2 index origin
OR 40.02  ; index right turn
AND 40.00  ; index right comm
OUT 40.02  ; index right turn
; rung 3
LD 0.01  ; LS2 index origin
OR 40.04  ; iindex right fin
AND 40.02  ; index right turn
OUT 40.04  ; iindex right fin
TIM 010 #3
; rung 4
LD TIM010  ; $?St$Bk?_#[87] / INDEX RIGTH END / $?St$Bk?_#[87]
AND 42.00  ; $?St$Bk?_#[69] / first cycle end / $?St$Bk?_#[69]
AND 34.04  ; work=1丄馨�1屄棳
AND 40.04  ; iindex right fin
OUT 40.06  ; rotary table not
; rung 5
LD TIM010  ; $?St$Bk?_#[87] / INDEX RIGTH END / $?St$Bk?_#[87]
OR 41.00  ; rotary table dow
AND 40.04  ; iindex right fin
OUT 41.00  ; rotary table dow
; rung 6
LD 3.01  ; LS8 ROTARY TABLE
OR 41.01  ; rotary table dow
AND 41.00  ; rotary table dow
OUT 41.01  ; rotary table dow

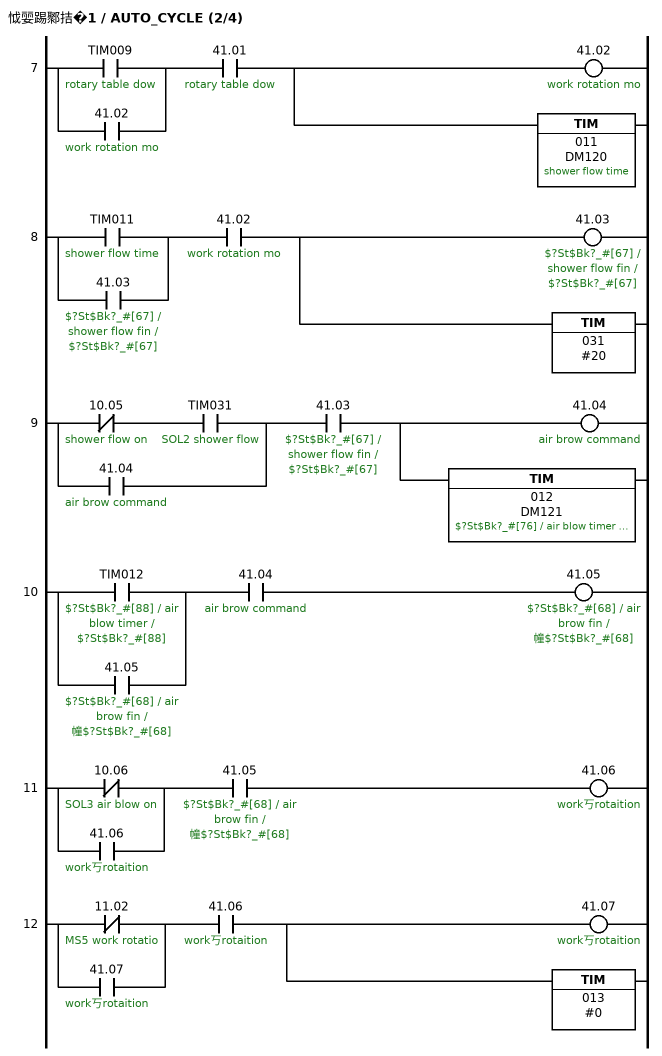
; rung 7
LD TIM009  ; rotary table dow
OR 41.02  ; work rotation mo
AND 41.01  ; rotary table dow
OUT 41.02  ; work rotation mo
TIM 011 DM120  ; shower flow time
; rung 8
LD TIM011  ; shower flow time
OR 41.03  ; $?St$Bk?_#[67] / shower flow fin / $?St$Bk?_#[67]
AND 41.02  ; work rotation mo
OUT 41.03  ; $?St$Bk?_#[67] / shower flow fin / $?St$Bk?_#[67]
TIM 031 #20
; rung 9
LDNOT 10.05  ; shower flow on
AND TIM031  ; SOL2 shower flow
OR 41.04  ; air brow command
AND 41.03  ; $?St$Bk?_#[67] / shower flow fin / $?St$Bk?_#[67]
OUT 41.04  ; air brow command
TIM 012 DM121  ; $?St$Bk?_#[76] / air blow timer / $?St$Bk?_#[76]
; rung 10
LD TIM012  ; $?St$Bk?_#[88] / air blow timer / $?St$Bk?_#[88]
OR 41.05  ; $?St$Bk?_#[68] / air brow fin / 幢$?St$Bk?_#[68]
AND 41.04  ; air brow command
OUT 41.05  ; $?St$Bk?_#[68] / air brow fin / 幢$?St$Bk?_#[68]
; rung 11
LDNOT 10.06  ; SOL3 air blow on
OR 41.06  ; work丂rotaition
AND 41.05  ; $?St$Bk?_#[68] / air brow fin / 幢$?St$Bk?_#[68]
OUT 41.06  ; work丂rotaition
; rung 12
LDNOT 11.02  ; MS5 work rotatio
OR 41.07  ; work丂rotaition
AND 41.06  ; work丂rotaition
OUT 41.07  ; work丂rotaition
TIM 013 #0

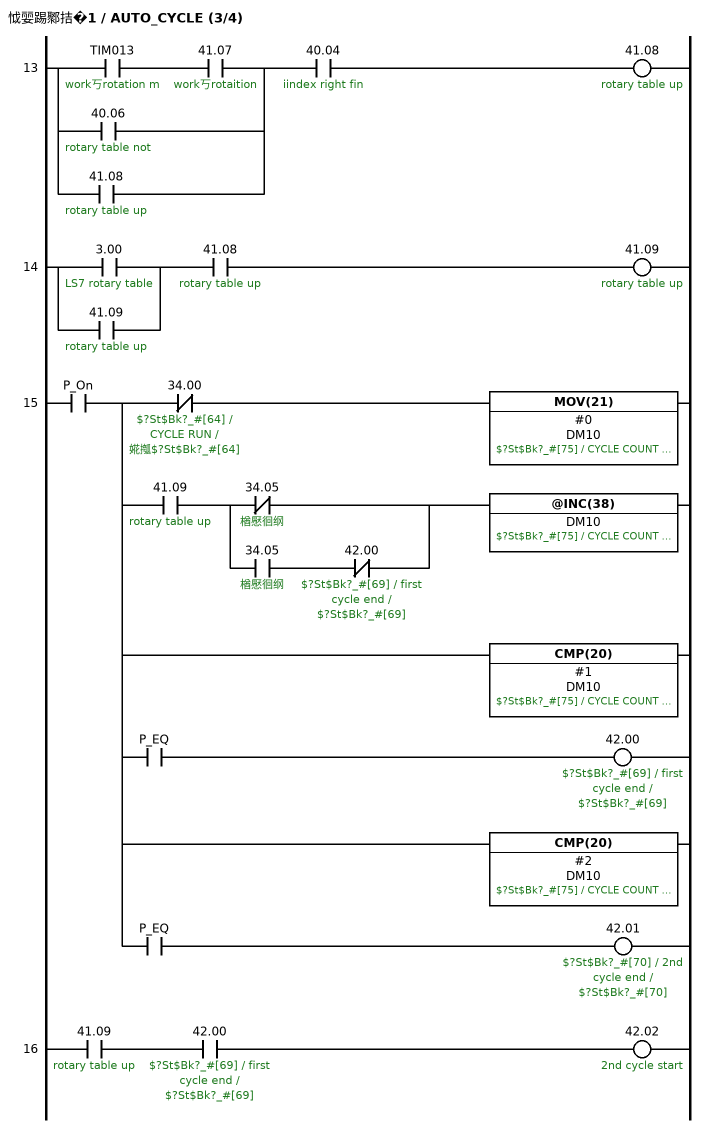
; rung 13
LD TIM013  ; work丂rotation m
AND 41.07  ; work丂rotaition
OR 40.06  ; rotary table not
OR 41.08  ; rotary table up
AND 40.04  ; iindex right fin
OUT 41.08  ; rotary table up
; rung 14
LD 3.00  ; LS7 rotary table
OR 41.09  ; rotary table up
AND 41.08  ; rotary table up
OUT 41.09  ; rotary table up
; rung 15
LD P_On
OUT TR0
ANDNOT 34.00  ; $?St$Bk?_#[64] / CYCLE RUN / 婲摦$?St$Bk?_#[64]
MOV(21) #0 DM10  ; $?St$Bk?_#[75] / CYCLE COUNT / 徊�$?St$Bk?_#[75]
LD TR0
AND 41.09  ; rotary table up
LDNOT 34.05  ; 楢懕徊纲
LD 34.05  ; 楢懕徊纲
ANDNOT 42.00  ; $?St$Bk?_#[69] / first cycle end / $?St$Bk?_#[69]
ORLD
ANDLD
@INC(38) DM10  ; $?St$Bk?_#[75] / CYCLE COUNT / 徊�$?St$Bk?_#[75]
LD TR0
CMP(20) #1 DM10  ; $?St$Bk?_#[75] / CYCLE COUNT / 徊�$?St$Bk?_#[75]
AND P_EQ
OUT 42.00  ; $?St$Bk?_#[69] / first cycle end / $?St$Bk?_#[69]
LD TR0
CMP(20) #2 DM10  ; $?St$Bk?_#[75] / CYCLE COUNT / 徊�$?St$Bk?_#[75]
AND P_EQ
OUT 42.01  ; $?St$Bk?_#[70] / 2nd cycle end / $?St$Bk?_#[70]
; rung 16
LD 41.09  ; rotary table up
AND 42.00  ; $?St$Bk?_#[69] / first cycle end / $?St$Bk?_#[69]
OUT 42.02  ; 2nd cycle start

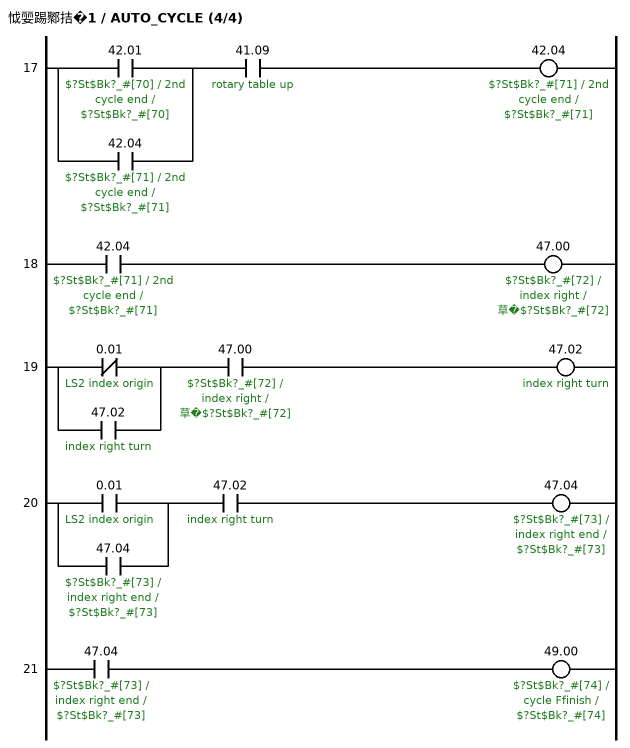
; rung 17
LD 42.01  ; $?St$Bk?_#[70] / 2nd cycle end / $?St$Bk?_#[70]
OR 42.04  ; $?St$Bk?_#[71] / 2nd cycle end / $?St$Bk?_#[71]
AND 41.09  ; rotary table up
OUT 42.04  ; $?St$Bk?_#[71] / 2nd cycle end / $?St$Bk?_#[71]
; rung 18
LD 42.04  ; $?St$Bk?_#[71] / 2nd cycle end / $?St$Bk?_#[71]
OUT 47.00  ; $?St$Bk?_#[72] / index right / 草�$?St$Bk?_#[72]
; rung 19
LDNOT 0.01  ; LS2 index origin
OR 47.02  ; index right turn
AND 47.00  ; $?St$Bk?_#[72] / index right / 草�$?St$Bk?_#[72]
OUT 47.02  ; index right turn
; rung 20
LD 0.01  ; LS2 index origin
OR 47.04  ; $?St$Bk?_#[73] / index right end / $?St$Bk?_#[73]
AND 47.02  ; index right turn
OUT 47.04  ; $?St$Bk?_#[73] / index right end / $?St$Bk?_#[73]
; rung 21
LD 47.04  ; $?St$Bk?_#[73] / index right end / $?St$Bk?_#[73]
OUT 49.00  ; $?St$Bk?_#[74] / cycle Ffinish / $?St$Bk?_#[74]

### Section MANUAL

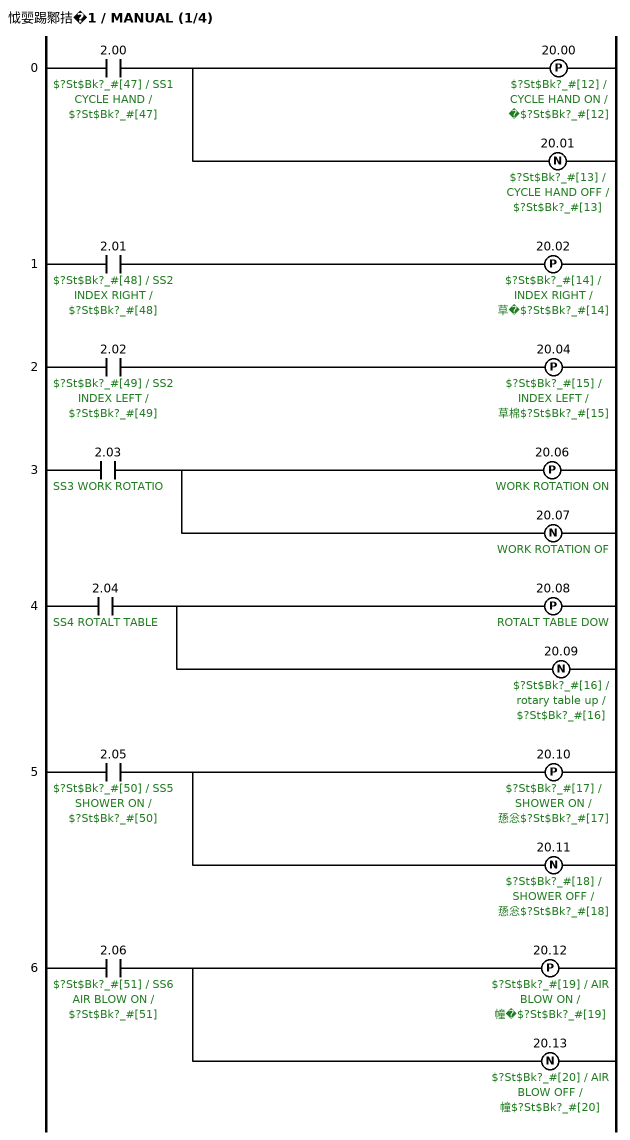
; rung 0
LD 2.00  ; $?St$Bk?_#[47] / SS1 CYCLE HAND / $?St$Bk?_#[47]
DIFU(13) 20.00  ; $?St$Bk?_#[12] / CYCLE HAND ON / �$?St$Bk?_#[12]
DIFD(14) 20.01  ; $?St$Bk?_#[13] / CYCLE HAND OFF / $?St$Bk?_#[13]
; rung 1
LD 2.01  ; $?St$Bk?_#[48] / SS2 INDEX RIGHT / $?St$Bk?_#[48]
DIFU(13) 20.02  ; $?St$Bk?_#[14] / INDEX RIGHT / 草�$?St$Bk?_#[14]
; rung 2
LD 2.02  ; $?St$Bk?_#[49] / SS2 INDEX LEFT / $?St$Bk?_#[49]
DIFU(13) 20.04  ; $?St$Bk?_#[15] / INDEX LEFT / 草棉$?St$Bk?_#[15]
; rung 3
LD 2.03  ; SS3 WORK ROTATIO
DIFU(13) 20.06  ; WORK ROTATION ON
DIFD(14) 20.07  ; WORK ROTATION OF
; rung 4
LD 2.04  ; SS4 ROTALT TABLE
DIFU(13) 20.08  ; ROTALT TABLE DOW
DIFD(14) 20.09  ; $?St$Bk?_#[16] / rotary table up / $?St$Bk?_#[16]
; rung 5
LD 2.05  ; $?St$Bk?_#[50] / SS5 SHOWER ON / $?St$Bk?_#[50]
DIFU(13) 20.10  ; $?St$Bk?_#[17] / SHOWER ON / 愻忩$?St$Bk?_#[17]
DIFD(14) 20.11  ; $?St$Bk?_#[18] / SHOWER OFF / 愻忩$?St$Bk?_#[18]
; rung 6
LD 2.06  ; $?St$Bk?_#[51] / SS6 AIR BLOW ON / $?St$Bk?_#[51]
DIFU(13) 20.12  ; $?St$Bk?_#[19] / AIR BLOW ON / 幢�$?St$Bk?_#[19]
DIFD(14) 20.13  ; $?St$Bk?_#[20] / AIR BLOW OFF / 幢$?St$Bk?_#[20]

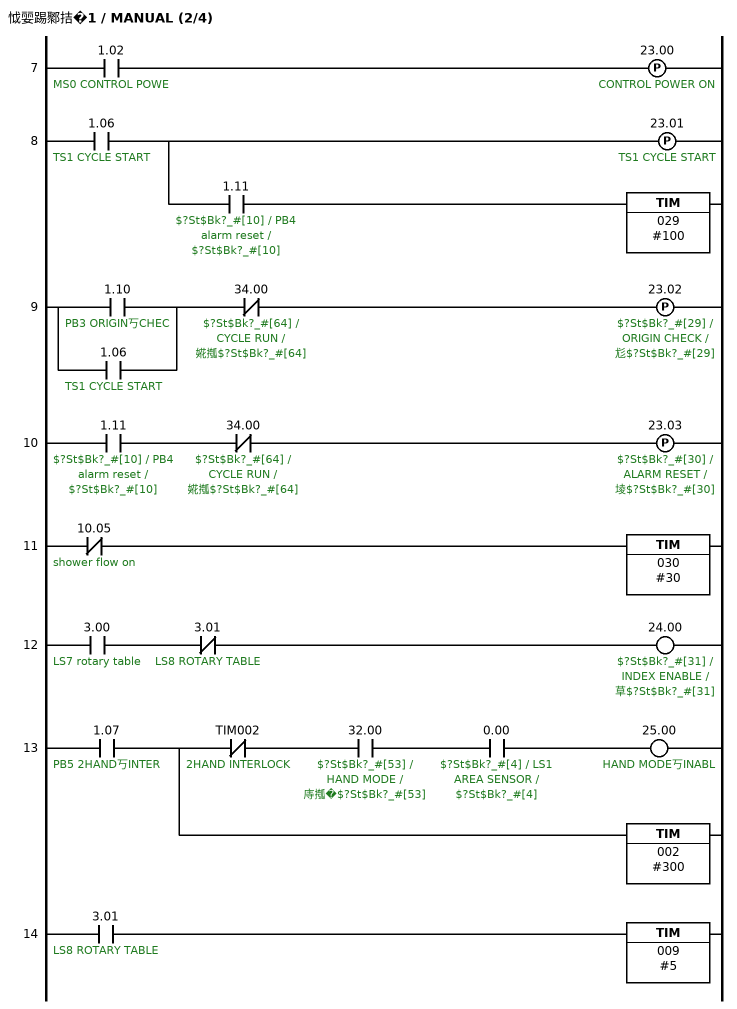
; rung 7
LD 1.02  ; MS0 CONTROL POWE
DIFU(13) 23.00  ; CONTROL POWER ON
; rung 8
LD 1.06  ; TS1 CYCLE START
DIFU(13) 23.01  ; TS1 CYCLE START
AND 1.11  ; $?St$Bk?_#[10] / PB4 alarm reset / $?St$Bk?_#[10]
TIM 029 #100
; rung 9
LD 1.10  ; PB3 ORIGIN丂CHEC
OR 1.06  ; TS1 CYCLE START
ANDNOT 34.00  ; $?St$Bk?_#[64] / CYCLE RUN / 婲摦$?St$Bk?_#[64]
DIFU(13) 23.02  ; $?St$Bk?_#[29] / ORIGIN CHECK / 尨$?St$Bk?_#[29]
; rung 10
LD 1.11  ; $?St$Bk?_#[10] / PB4 alarm reset / $?St$Bk?_#[10]
ANDNOT 34.00  ; $?St$Bk?_#[64] / CYCLE RUN / 婲摦$?St$Bk?_#[64]
DIFU(13) 23.03  ; $?St$Bk?_#[30] / ALARM RESET / 堎$?St$Bk?_#[30]
; rung 11
LDNOT 10.05  ; shower flow on
TIM 030 #30
; rung 12
LD 3.00  ; LS7 rotary table
ANDNOT 3.01  ; LS8 ROTARY TABLE
OUT 24.00  ; $?St$Bk?_#[31] / INDEX ENABLE / 草$?St$Bk?_#[31]
; rung 13
LD 1.07  ; PB5 2HAND丂INTER
OUT TR0
ANDNOT TIM002  ; 2HAND INTERLOCK
AND 32.00  ; $?St$Bk?_#[53] / HAND MODE / 庤摦�$?St$Bk?_#[53]
AND 0.00  ; $?St$Bk?_#[4] / LS1 AREA SENSOR / $?St$Bk?_#[4]
OUT 25.00  ; HAND MODE丂INABL
LD TR0
TIM 002 #300
; rung 14
LD 3.01  ; LS8 ROTARY TABLE
TIM 009 #5

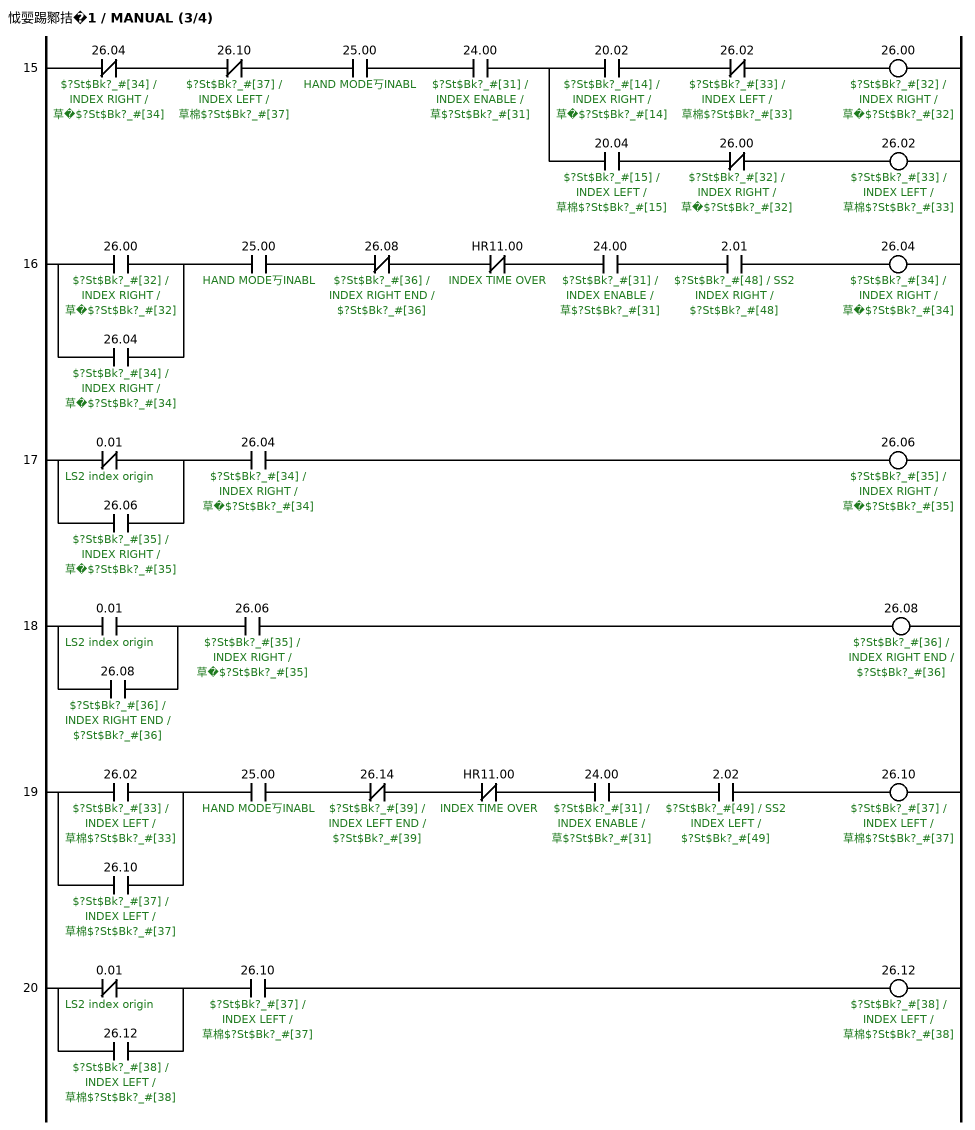
; rung 15
LDNOT 26.04  ; $?St$Bk?_#[34] / INDEX RIGHT / 草�$?St$Bk?_#[34]
ANDNOT 26.10  ; $?St$Bk?_#[37] / INDEX LEFT / 草棉$?St$Bk?_#[37]
AND 25.00  ; HAND MODE丂INABL
AND 24.00  ; $?St$Bk?_#[31] / INDEX ENABLE / 草$?St$Bk?_#[31]
OUT TR0
AND 20.02  ; $?St$Bk?_#[14] / INDEX RIGHT / 草�$?St$Bk?_#[14]
ANDNOT 26.02  ; $?St$Bk?_#[33] / INDEX LEFT / 草棉$?St$Bk?_#[33]
OUT 26.00  ; $?St$Bk?_#[32] / INDEX RIGHT / 草�$?St$Bk?_#[32]
LD TR0
AND 20.04  ; $?St$Bk?_#[15] / INDEX LEFT / 草棉$?St$Bk?_#[15]
ANDNOT 26.00  ; $?St$Bk?_#[32] / INDEX RIGHT / 草�$?St$Bk?_#[32]
OUT 26.02  ; $?St$Bk?_#[33] / INDEX LEFT / 草棉$?St$Bk?_#[33]
; rung 16
LD 26.00  ; $?St$Bk?_#[32] / INDEX RIGHT / 草�$?St$Bk?_#[32]
OR 26.04  ; $?St$Bk?_#[34] / INDEX RIGHT / 草�$?St$Bk?_#[34]
AND 25.00  ; HAND MODE丂INABL
ANDNOT 26.08  ; $?St$Bk?_#[36] / INDEX RIGHT END / $?St$Bk?_#[36]
ANDNOT HR11.00  ; INDEX TIME OVER
AND 24.00  ; $?St$Bk?_#[31] / INDEX ENABLE / 草$?St$Bk?_#[31]
AND 2.01  ; $?St$Bk?_#[48] / SS2 INDEX RIGHT / $?St$Bk?_#[48]
OUT 26.04  ; $?St$Bk?_#[34] / INDEX RIGHT / 草�$?St$Bk?_#[34]
; rung 17
LDNOT 0.01  ; LS2 index origin
OR 26.06  ; $?St$Bk?_#[35] / INDEX RIGHT / 草�$?St$Bk?_#[35]
AND 26.04  ; $?St$Bk?_#[34] / INDEX RIGHT / 草�$?St$Bk?_#[34]
OUT 26.06  ; $?St$Bk?_#[35] / INDEX RIGHT / 草�$?St$Bk?_#[35]
; rung 18
LD 0.01  ; LS2 index origin
OR 26.08  ; $?St$Bk?_#[36] / INDEX RIGHT END / $?St$Bk?_#[36]
AND 26.06  ; $?St$Bk?_#[35] / INDEX RIGHT / 草�$?St$Bk?_#[35]
OUT 26.08  ; $?St$Bk?_#[36] / INDEX RIGHT END / $?St$Bk?_#[36]
; rung 19
LD 26.02  ; $?St$Bk?_#[33] / INDEX LEFT / 草棉$?St$Bk?_#[33]
OR 26.10  ; $?St$Bk?_#[37] / INDEX LEFT / 草棉$?St$Bk?_#[37]
AND 25.00  ; HAND MODE丂INABL
ANDNOT 26.14  ; $?St$Bk?_#[39] / INDEX LEFT END / $?St$Bk?_#[39]
ANDNOT HR11.00  ; INDEX TIME OVER
AND 24.00  ; $?St$Bk?_#[31] / INDEX ENABLE / 草$?St$Bk?_#[31]
AND 2.02  ; $?St$Bk?_#[49] / SS2 INDEX LEFT / $?St$Bk?_#[49]
OUT 26.10  ; $?St$Bk?_#[37] / INDEX LEFT / 草棉$?St$Bk?_#[37]
; rung 20
LDNOT 0.01  ; LS2 index origin
OR 26.12  ; $?St$Bk?_#[38] / INDEX LEFT / 草棉$?St$Bk?_#[38]
AND 26.10  ; $?St$Bk?_#[37] / INDEX LEFT / 草棉$?St$Bk?_#[37]
OUT 26.12  ; $?St$Bk?_#[38] / INDEX LEFT / 草棉$?St$Bk?_#[38]

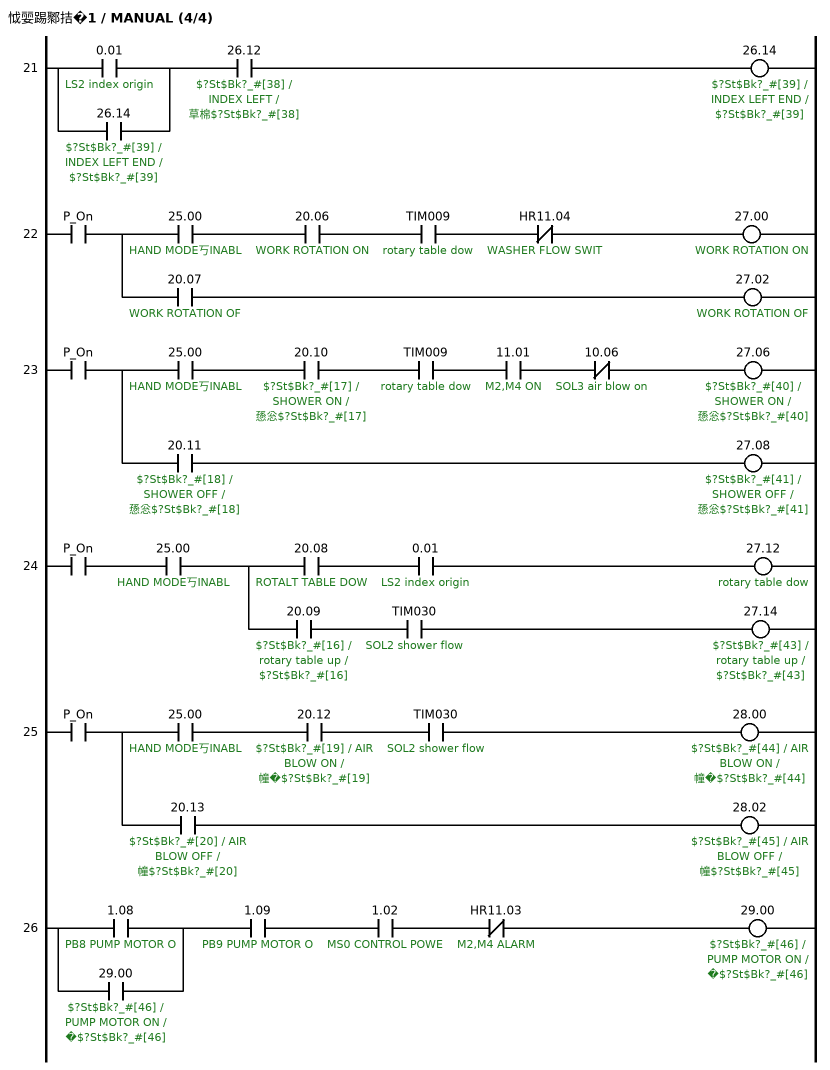
; rung 21
LD 0.01  ; LS2 index origin
OR 26.14  ; $?St$Bk?_#[39] / INDEX LEFT END / $?St$Bk?_#[39]
AND 26.12  ; $?St$Bk?_#[38] / INDEX LEFT / 草棉$?St$Bk?_#[38]
OUT 26.14  ; $?St$Bk?_#[39] / INDEX LEFT END / $?St$Bk?_#[39]
; rung 22
LD P_On
OUT TR0
AND 25.00  ; HAND MODE丂INABL
AND 20.06  ; WORK ROTATION ON
AND TIM009  ; rotary table dow
ANDNOT HR11.04  ; WASHER FLOW SWIT
OUT 27.00  ; WORK ROTATION ON
LD TR0
AND 20.07  ; WORK ROTATION OF
OUT 27.02  ; WORK ROTATION OF
; rung 23
LD P_On
OUT TR0
AND 25.00  ; HAND MODE丂INABL
AND 20.10  ; $?St$Bk?_#[17] / SHOWER ON / 愻忩$?St$Bk?_#[17]
AND TIM009  ; rotary table dow
AND 11.01  ; M2,M4 ON
ANDNOT 10.06  ; SOL3 air blow on
OUT 27.06  ; $?St$Bk?_#[40] / SHOWER ON / 愻忩$?St$Bk?_#[40]
LD TR0
AND 20.11  ; $?St$Bk?_#[18] / SHOWER OFF / 愻忩$?St$Bk?_#[18]
OUT 27.08  ; $?St$Bk?_#[41] / SHOWER OFF / 愻忩$?St$Bk?_#[41]
; rung 24
LD P_On
AND 25.00  ; HAND MODE丂INABL
OUT TR0
AND 20.08  ; ROTALT TABLE DOW
AND 0.01  ; LS2 index origin
OUT 27.12  ; rotary table dow
LD TR0
AND 20.09  ; $?St$Bk?_#[16] / rotary table up / $?St$Bk?_#[16]
AND TIM030  ; SOL2 shower flow
OUT 27.14  ; $?St$Bk?_#[43] / rotary table up / $?St$Bk?_#[43]
; rung 25
LD P_On
OUT TR0
AND 25.00  ; HAND MODE丂INABL
AND 20.12  ; $?St$Bk?_#[19] / AIR BLOW ON / 幢�$?St$Bk?_#[19]
AND TIM030  ; SOL2 shower flow
OUT 28.00  ; $?St$Bk?_#[44] / AIR BLOW ON / 幢�$?St$Bk?_#[44]
LD TR0
AND 20.13  ; $?St$Bk?_#[20] / AIR BLOW OFF / 幢$?St$Bk?_#[20]
OUT 28.02  ; $?St$Bk?_#[45] / AIR BLOW OFF / 幢$?St$Bk?_#[45]
; rung 26
LD 1.08  ; PB8 PUMP MOTOR O
OR 29.00  ; $?St$Bk?_#[46] / PUMP MOTOR ON / �$?St$Bk?_#[46]
AND 1.09  ; PB9 PUMP MOTOR O
AND 1.02  ; MS0 CONTROL POWE
ANDNOT HR11.03  ; M2,M4 ALARM
OUT 29.00  ; $?St$Bk?_#[46] / PUMP MOTOR ON / �$?St$Bk?_#[46]

### Section MANUAL1

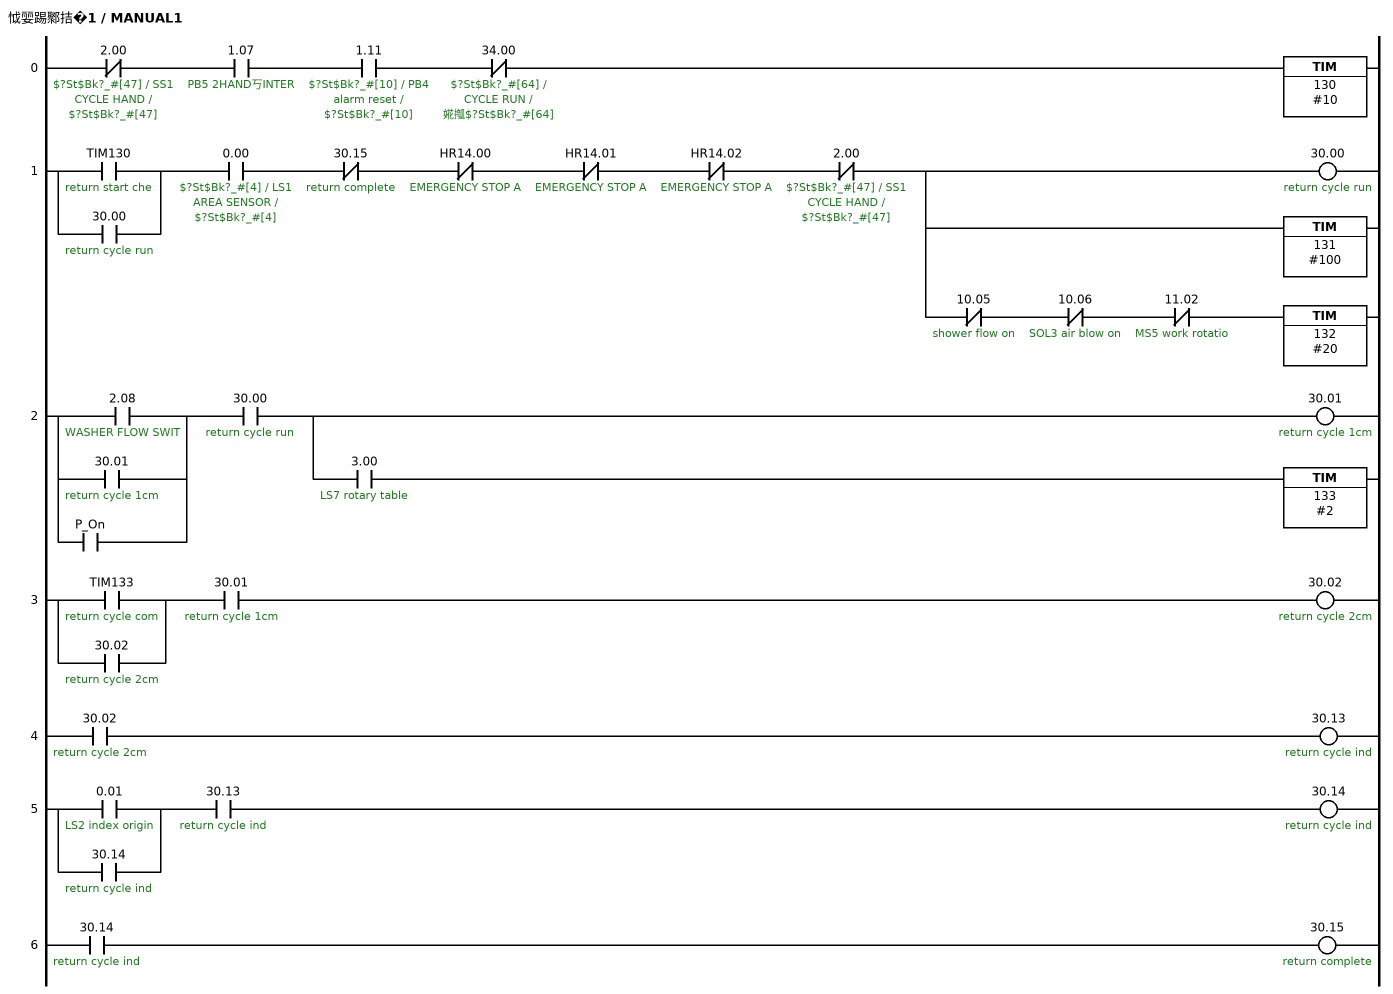
; rung 0
LDNOT 2.00  ; $?St$Bk?_#[47] / SS1 CYCLE HAND / $?St$Bk?_#[47]
AND 1.07  ; PB5 2HAND丂INTER
AND 1.11  ; $?St$Bk?_#[10] / PB4 alarm reset / $?St$Bk?_#[10]
ANDNOT 34.00  ; $?St$Bk?_#[64] / CYCLE RUN / 婲摦$?St$Bk?_#[64]
TIM 130 #10
; rung 1
LD TIM130  ; return start che
OR 30.00  ; return cycle run
AND 0.00  ; $?St$Bk?_#[4] / LS1 AREA SENSOR / $?St$Bk?_#[4]
ANDNOT 30.15  ; return complete
ANDNOT HR14.00  ; EMERGENCY STOP A
ANDNOT HR14.01  ; EMERGENCY STOP A
ANDNOT HR14.02  ; EMERGENCY STOP A
ANDNOT 2.00  ; $?St$Bk?_#[47] / SS1 CYCLE HAND / $?St$Bk?_#[47]
OUT 30.00  ; return cycle run
TIM 131 #100
ANDNOT 10.05  ; shower flow on
ANDNOT 10.06  ; SOL3 air blow on
ANDNOT 11.02  ; MS5 work rotatio
TIM 132 #20
; rung 2
LD 2.08  ; WASHER FLOW SWIT
OR 30.01  ; return cycle 1cm
OR P_On
AND 30.00  ; return cycle run
OUT 30.01  ; return cycle 1cm
AND 3.00  ; LS7 rotary table
TIM 133 #2
; rung 3
LD TIM133  ; return cycle com
OR 30.02  ; return cycle 2cm
AND 30.01  ; return cycle 1cm
OUT 30.02  ; return cycle 2cm
; rung 4
LD 30.02  ; return cycle 2cm
OUT 30.13  ; return cycle ind
; rung 5
LD 0.01  ; LS2 index origin
OR 30.14  ; return cycle ind
AND 30.13  ; return cycle ind
OUT 30.14  ; return cycle ind
; rung 6
LD 30.14  ; return cycle ind
OUT 30.15  ; return complete

### Section OUTPUT

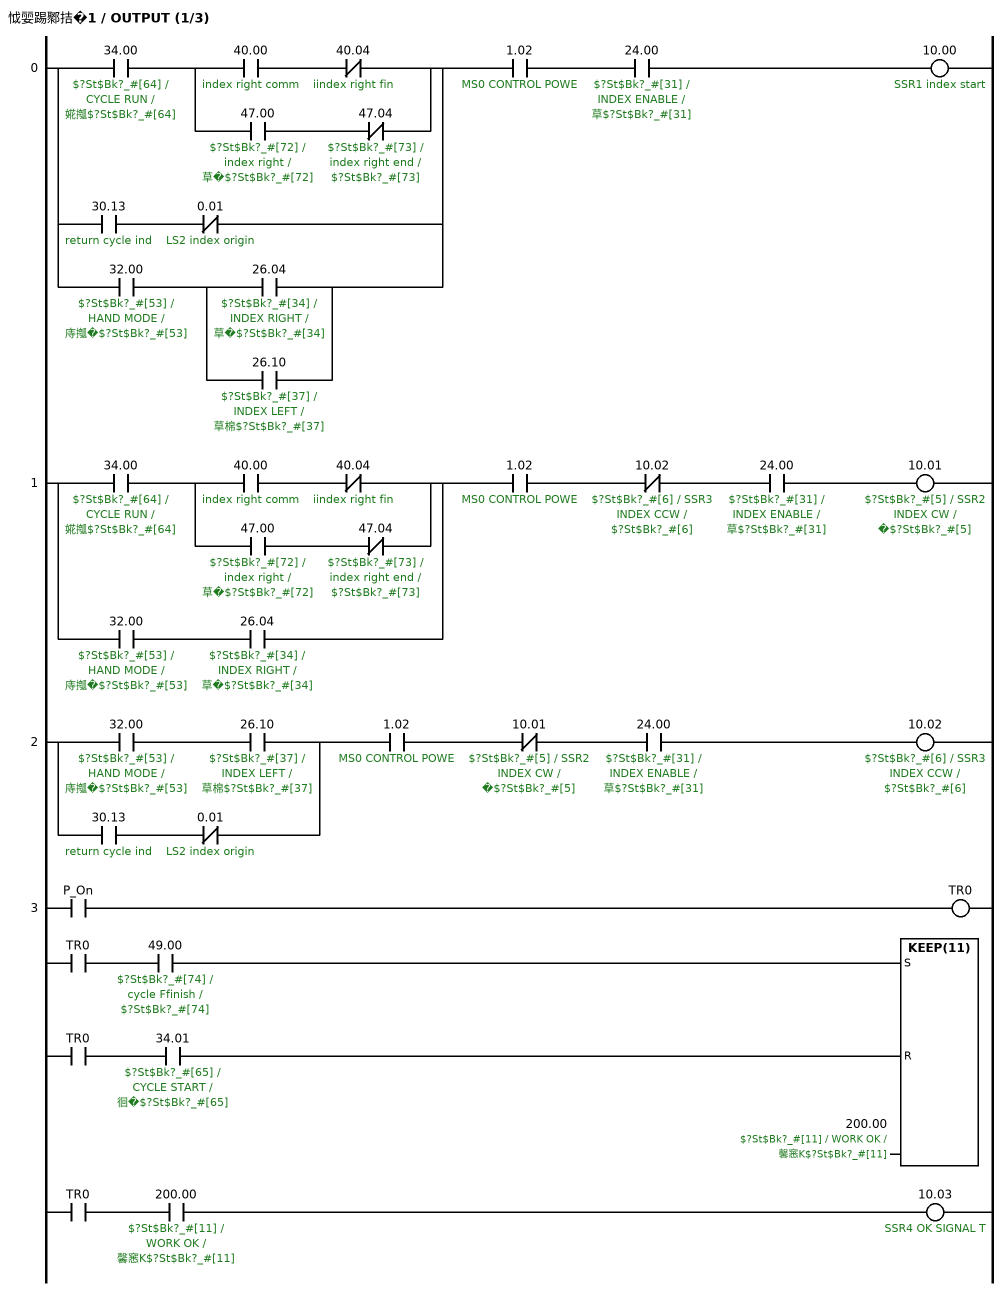
; rung 0
LD 34.00  ; $?St$Bk?_#[64] / CYCLE RUN / 婲摦$?St$Bk?_#[64]
LD 40.00  ; index right comm
ANDNOT 40.04  ; iindex right fin
LD 47.00  ; $?St$Bk?_#[72] / index right / 草�$?St$Bk?_#[72]
ANDNOT 47.04  ; $?St$Bk?_#[73] / index right end / $?St$Bk?_#[73]
ORLD
ANDLD
LD 30.13  ; return cycle ind
ANDNOT 0.01  ; LS2 index origin
ORLD
LD 32.00  ; $?St$Bk?_#[53] / HAND MODE / 庤摦�$?St$Bk?_#[53]
LD 26.04  ; $?St$Bk?_#[34] / INDEX RIGHT / 草�$?St$Bk?_#[34]
OR 26.10  ; $?St$Bk?_#[37] / INDEX LEFT / 草棉$?St$Bk?_#[37]
ANDLD
ORLD
AND 1.02  ; MS0 CONTROL POWE
AND 24.00  ; $?St$Bk?_#[31] / INDEX ENABLE / 草$?St$Bk?_#[31]
OUT 10.00  ; SSR1 index start
; rung 1
LD 34.00  ; $?St$Bk?_#[64] / CYCLE RUN / 婲摦$?St$Bk?_#[64]
LD 40.00  ; index right comm
ANDNOT 40.04  ; iindex right fin
LD 47.00  ; $?St$Bk?_#[72] / index right / 草�$?St$Bk?_#[72]
ANDNOT 47.04  ; $?St$Bk?_#[73] / index right end / $?St$Bk?_#[73]
ORLD
ANDLD
LD 32.00  ; $?St$Bk?_#[53] / HAND MODE / 庤摦�$?St$Bk?_#[53]
AND 26.04  ; $?St$Bk?_#[34] / INDEX RIGHT / 草�$?St$Bk?_#[34]
ORLD
AND 1.02  ; MS0 CONTROL POWE
ANDNOT 10.02  ; $?St$Bk?_#[6] / SSR3 INDEX CCW / $?St$Bk?_#[6]
AND 24.00  ; $?St$Bk?_#[31] / INDEX ENABLE / 草$?St$Bk?_#[31]
OUT 10.01  ; $?St$Bk?_#[5] / SSR2 INDEX CW / �$?St$Bk?_#[5]
; rung 2
LD 32.00  ; $?St$Bk?_#[53] / HAND MODE / 庤摦�$?St$Bk?_#[53]
AND 26.10  ; $?St$Bk?_#[37] / INDEX LEFT / 草棉$?St$Bk?_#[37]
LD 30.13  ; return cycle ind
ANDNOT 0.01  ; LS2 index origin
ORLD
AND 1.02  ; MS0 CONTROL POWE
ANDNOT 10.01  ; $?St$Bk?_#[5] / SSR2 INDEX CW / �$?St$Bk?_#[5]
AND 24.00  ; $?St$Bk?_#[31] / INDEX ENABLE / 草$?St$Bk?_#[31]
OUT 10.02  ; $?St$Bk?_#[6] / SSR3 INDEX CCW / $?St$Bk?_#[6]
; rung 3
LD P_On
OUT TR0
AND 49.00  ; $?St$Bk?_#[74] / cycle Ffinish / $?St$Bk?_#[74]
LD TR0
AND 34.01  ; $?St$Bk?_#[65] / CYCLE START / 徊�$?St$Bk?_#[65]
KEEP(11) 200.00  ; $?St$Bk?_#[11] / WORK OK / 馨窸K$?St$Bk?_#[11]
LD TR0
AND 200.00  ; $?St$Bk?_#[11] / WORK OK / 馨窸K$?St$Bk?_#[11]
OUT 10.03  ; SSR4 OK SIGNAL T

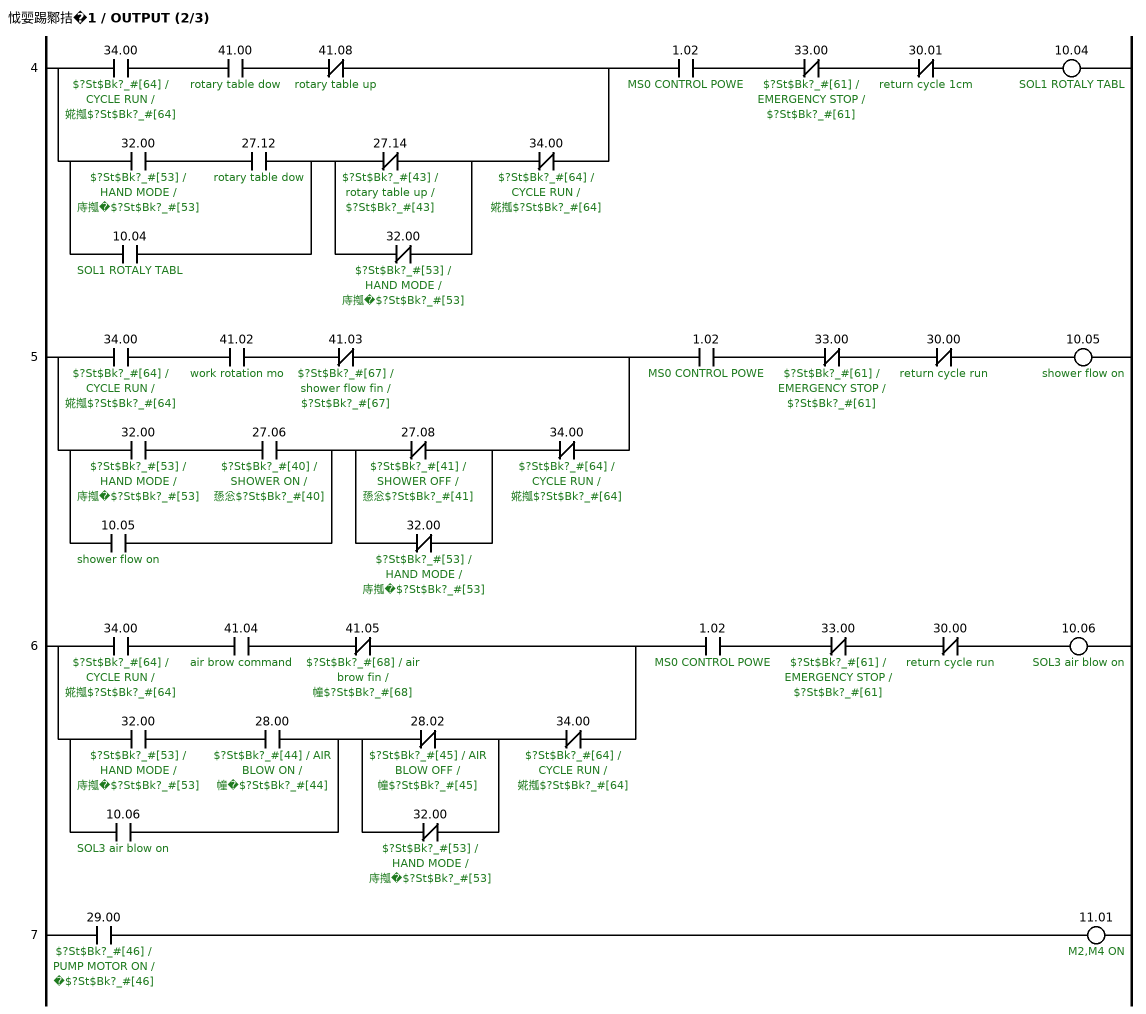
; rung 4
LD 34.00  ; $?St$Bk?_#[64] / CYCLE RUN / 婲摦$?St$Bk?_#[64]
AND 41.00  ; rotary table dow
ANDNOT 41.08  ; rotary table up
LD 32.00  ; $?St$Bk?_#[53] / HAND MODE / 庤摦�$?St$Bk?_#[53]
AND 27.12  ; rotary table dow
OR 10.04  ; SOL1 ROTALY TABL
LDNOT 27.14  ; $?St$Bk?_#[43] / rotary table up / $?St$Bk?_#[43]
ORNOT 32.00  ; $?St$Bk?_#[53] / HAND MODE / 庤摦�$?St$Bk?_#[53]
ANDLD
ANDNOT 34.00  ; $?St$Bk?_#[64] / CYCLE RUN / 婲摦$?St$Bk?_#[64]
ORLD
AND 1.02  ; MS0 CONTROL POWE
ANDNOT 33.00  ; $?St$Bk?_#[61] / EMERGENCY STOP / $?St$Bk?_#[61]
ANDNOT 30.01  ; return cycle 1cm
OUT 10.04  ; SOL1 ROTALY TABL
; rung 5
LD 34.00  ; $?St$Bk?_#[64] / CYCLE RUN / 婲摦$?St$Bk?_#[64]
AND 41.02  ; work rotation mo
ANDNOT 41.03  ; $?St$Bk?_#[67] / shower flow fin / $?St$Bk?_#[67]
LD 32.00  ; $?St$Bk?_#[53] / HAND MODE / 庤摦�$?St$Bk?_#[53]
AND 27.06  ; $?St$Bk?_#[40] / SHOWER ON / 愻忩$?St$Bk?_#[40]
OR 10.05  ; shower flow on
LDNOT 27.08  ; $?St$Bk?_#[41] / SHOWER OFF / 愻忩$?St$Bk?_#[41]
ORNOT 32.00  ; $?St$Bk?_#[53] / HAND MODE / 庤摦�$?St$Bk?_#[53]
ANDLD
ANDNOT 34.00  ; $?St$Bk?_#[64] / CYCLE RUN / 婲摦$?St$Bk?_#[64]
ORLD
AND 1.02  ; MS0 CONTROL POWE
ANDNOT 33.00  ; $?St$Bk?_#[61] / EMERGENCY STOP / $?St$Bk?_#[61]
ANDNOT 30.00  ; return cycle run
OUT 10.05  ; shower flow on
; rung 6
LD 34.00  ; $?St$Bk?_#[64] / CYCLE RUN / 婲摦$?St$Bk?_#[64]
AND 41.04  ; air brow command
ANDNOT 41.05  ; $?St$Bk?_#[68] / air brow fin / 幢$?St$Bk?_#[68]
LD 32.00  ; $?St$Bk?_#[53] / HAND MODE / 庤摦�$?St$Bk?_#[53]
AND 28.00  ; $?St$Bk?_#[44] / AIR BLOW ON / 幢�$?St$Bk?_#[44]
OR 10.06  ; SOL3 air blow on
LDNOT 28.02  ; $?St$Bk?_#[45] / AIR BLOW OFF / 幢$?St$Bk?_#[45]
ORNOT 32.00  ; $?St$Bk?_#[53] / HAND MODE / 庤摦�$?St$Bk?_#[53]
ANDLD
ANDNOT 34.00  ; $?St$Bk?_#[64] / CYCLE RUN / 婲摦$?St$Bk?_#[64]
ORLD
AND 1.02  ; MS0 CONTROL POWE
ANDNOT 33.00  ; $?St$Bk?_#[61] / EMERGENCY STOP / $?St$Bk?_#[61]
ANDNOT 30.00  ; return cycle run
OUT 10.06  ; SOL3 air blow on
; rung 7
LD 29.00  ; $?St$Bk?_#[46] / PUMP MOTOR ON / �$?St$Bk?_#[46]
OUT 11.01  ; M2,M4 ON

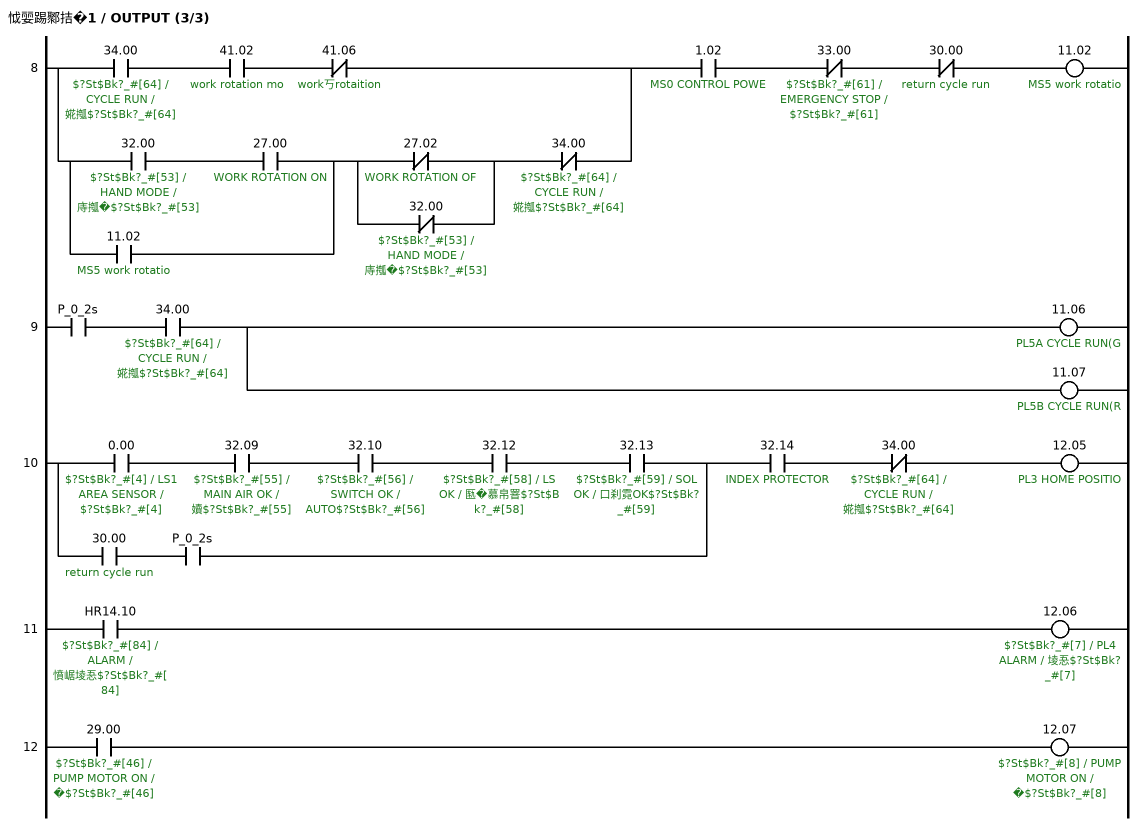
; rung 8
LD 34.00  ; $?St$Bk?_#[64] / CYCLE RUN / 婲摦$?St$Bk?_#[64]
AND 41.02  ; work rotation mo
ANDNOT 41.06  ; work丂rotaition
LD 32.00  ; $?St$Bk?_#[53] / HAND MODE / 庤摦�$?St$Bk?_#[53]
AND 27.00  ; WORK ROTATION ON
OR 11.02  ; MS5 work rotatio
LDNOT 27.02  ; WORK ROTATION OF
ORNOT 32.00  ; $?St$Bk?_#[53] / HAND MODE / 庤摦�$?St$Bk?_#[53]
ANDLD
ANDNOT 34.00  ; $?St$Bk?_#[64] / CYCLE RUN / 婲摦$?St$Bk?_#[64]
ORLD
AND 1.02  ; MS0 CONTROL POWE
ANDNOT 33.00  ; $?St$Bk?_#[61] / EMERGENCY STOP / $?St$Bk?_#[61]
ANDNOT 30.00  ; return cycle run
OUT 11.02  ; MS5 work rotatio
; rung 9
LD P_0_2s
AND 34.00  ; $?St$Bk?_#[64] / CYCLE RUN / 婲摦$?St$Bk?_#[64]
OUT 11.06  ; PL5A CYCLE RUN(G
OUT 11.07  ; PL5B CYCLE RUN(R
; rung 10
LD 0.00  ; $?St$Bk?_#[4] / LS1 AREA SENSOR / $?St$Bk?_#[4]
AND 32.09  ; $?St$Bk?_#[55] / MAIN AIR OK / 嬻$?St$Bk?_#[55]
AND 32.10  ; $?St$Bk?_#[56] / SWITCH OK / AUTO$?St$Bk?_#[56]
AND 32.12  ; $?St$Bk?_#[58] / LS OK / 匦�慕帛罯$?St$Bk?_#[58]
AND 32.13  ; $?St$Bk?_#[59] / SOL OK / 口刹霓OK$?St$Bk?_#[59]
LD 30.00  ; return cycle run
AND P_0_2s
ORLD
AND 32.14  ; INDEX PROTECTOR
ANDNOT 34.00  ; $?St$Bk?_#[64] / CYCLE RUN / 婲摦$?St$Bk?_#[64]
OUT 12.05  ; PL3 HOME POSITIO
; rung 11
LD HR14.10  ; $?St$Bk?_#[84] / ALARM / 憤崌堎忢$?St$Bk?_#[84]
OUT 12.06  ; $?St$Bk?_#[7] / PL4 ALARM / 堎忢$?St$Bk?_#[7]
; rung 12
LD 29.00  ; $?St$Bk?_#[46] / PUMP MOTOR ON / �$?St$Bk?_#[46]
OUT 12.07  ; $?St$Bk?_#[8] / PUMP MOTOR ON / �$?St$Bk?_#[8]

### Section MESSAGE

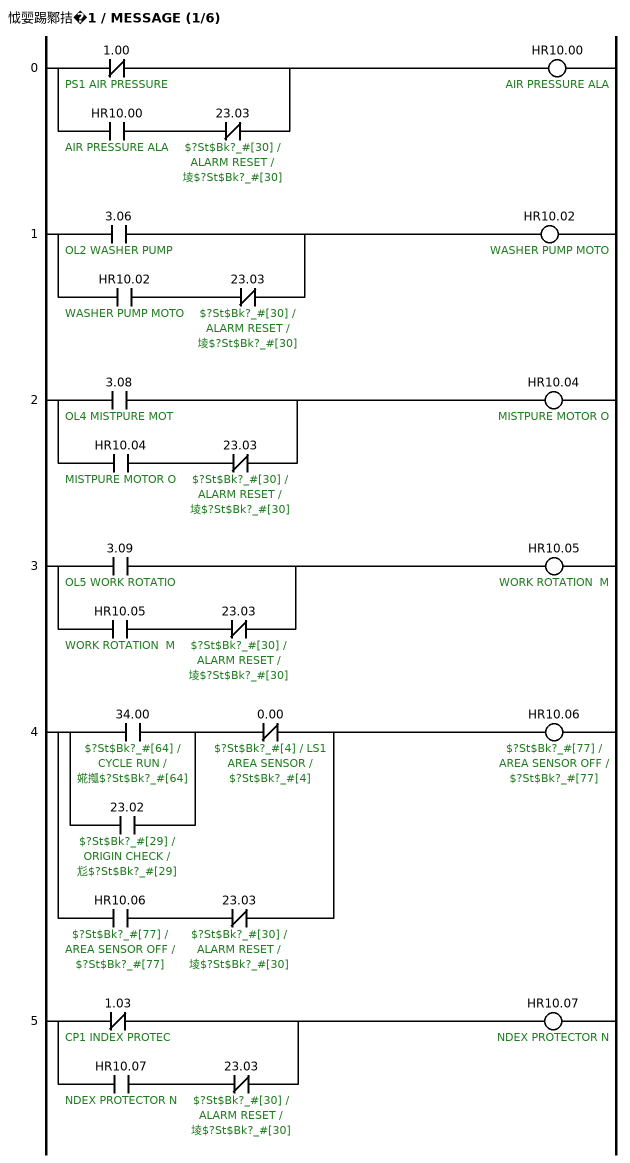
; rung 0
LDNOT 1.00  ; PS1 AIR PRESSURE
LD HR10.00  ; AIR PRESSURE ALA
ANDNOT 23.03  ; $?St$Bk?_#[30] / ALARM RESET / 堎$?St$Bk?_#[30]
ORLD
OUT HR10.00  ; AIR PRESSURE ALA
; rung 1
LD 3.06  ; OL2 WASHER PUMP
LD HR10.02  ; WASHER PUMP MOTO
ANDNOT 23.03  ; $?St$Bk?_#[30] / ALARM RESET / 堎$?St$Bk?_#[30]
ORLD
OUT HR10.02  ; WASHER PUMP MOTO
; rung 2
LD 3.08  ; OL4 MISTPURE MOT
LD HR10.04  ; MISTPURE MOTOR O
ANDNOT 23.03  ; $?St$Bk?_#[30] / ALARM RESET / 堎$?St$Bk?_#[30]
ORLD
OUT HR10.04  ; MISTPURE MOTOR O
; rung 3
LD 3.09  ; OL5 WORK ROTATIO
LD HR10.05  ; WORK ROTATION  M
ANDNOT 23.03  ; $?St$Bk?_#[30] / ALARM RESET / 堎$?St$Bk?_#[30]
ORLD
OUT HR10.05  ; WORK ROTATION  M
; rung 4
LD 34.00  ; $?St$Bk?_#[64] / CYCLE RUN / 婲摦$?St$Bk?_#[64]
OR 23.02  ; $?St$Bk?_#[29] / ORIGIN CHECK / 尨$?St$Bk?_#[29]
ANDNOT 0.00  ; $?St$Bk?_#[4] / LS1 AREA SENSOR / $?St$Bk?_#[4]
LD HR10.06  ; $?St$Bk?_#[77] / AREA SENSOR OFF / $?St$Bk?_#[77]
ANDNOT 23.03  ; $?St$Bk?_#[30] / ALARM RESET / 堎$?St$Bk?_#[30]
ORLD
OUT HR10.06  ; $?St$Bk?_#[77] / AREA SENSOR OFF / $?St$Bk?_#[77]
; rung 5
LDNOT 1.03  ; CP1 INDEX PROTEC
LD HR10.07  ; NDEX PROTECTOR N
ANDNOT 23.03  ; $?St$Bk?_#[30] / ALARM RESET / 堎$?St$Bk?_#[30]
ORLD
OUT HR10.07  ; NDEX PROTECTOR N

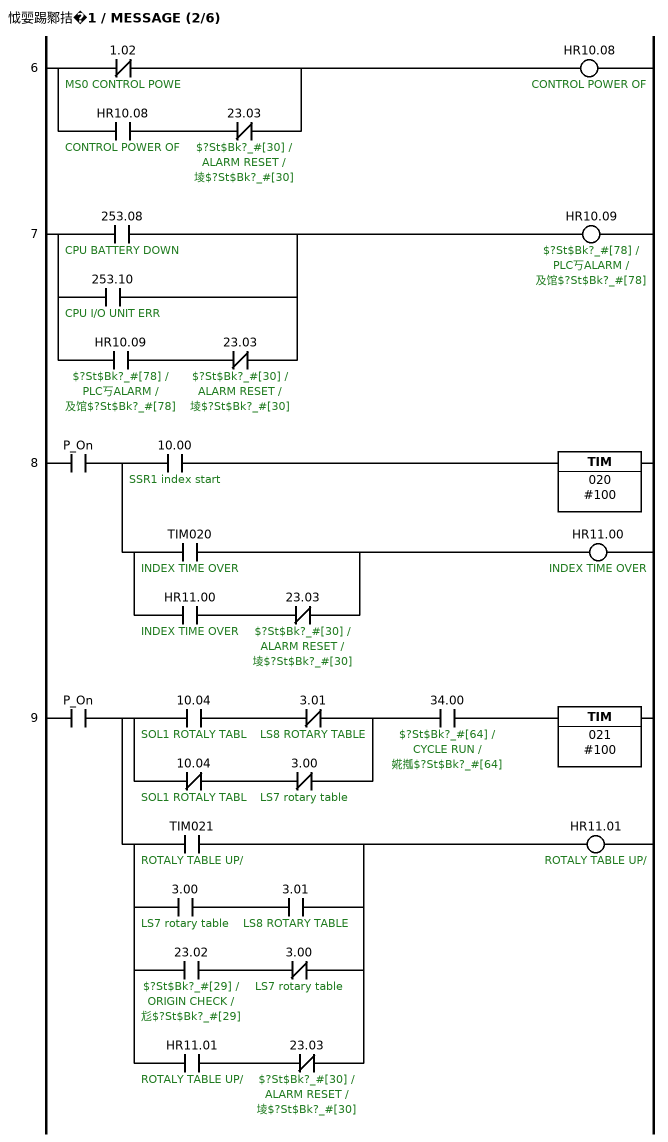
; rung 6
LDNOT 1.02  ; MS0 CONTROL POWE
LD HR10.08  ; CONTROL POWER OF
ANDNOT 23.03  ; $?St$Bk?_#[30] / ALARM RESET / 堎$?St$Bk?_#[30]
ORLD
OUT HR10.08  ; CONTROL POWER OF
; rung 7
LD 253.08  ; CPU BATTERY DOWN
OR 253.10  ; CPU I/O UNIT ERR
LD HR10.09  ; $?St$Bk?_#[78] / PLC丂ALARM / 及馆$?St$Bk?_#[78]
ANDNOT 23.03  ; $?St$Bk?_#[30] / ALARM RESET / 堎$?St$Bk?_#[30]
ORLD
OUT HR10.09  ; $?St$Bk?_#[78] / PLC丂ALARM / 及馆$?St$Bk?_#[78]
; rung 8
LD P_On
OUT TR0
AND 10.00  ; SSR1 index start
TIM 020 #100
LD TR0
LD TIM020  ; INDEX TIME OVER
LD HR11.00  ; INDEX TIME OVER
ANDNOT 23.03  ; $?St$Bk?_#[30] / ALARM RESET / 堎$?St$Bk?_#[30]
ORLD
ANDLD
OUT HR11.00  ; INDEX TIME OVER
; rung 9
LD P_On
OUT TR0
LD 10.04  ; SOL1 ROTALY TABL
ANDNOT 3.01  ; LS8 ROTARY TABLE
LDNOT 10.04  ; SOL1 ROTALY TABL
ANDNOT 3.00  ; LS7 rotary table
ORLD
ANDLD
AND 34.00  ; $?St$Bk?_#[64] / CYCLE RUN / 婲摦$?St$Bk?_#[64]
TIM 021 #100
LD TR0
LD TIM021  ; ROTALY TABLE UP/
LD 3.00  ; LS7 rotary table
AND 3.01  ; LS8 ROTARY TABLE
ORLD
LD 23.02  ; $?St$Bk?_#[29] / ORIGIN CHECK / 尨$?St$Bk?_#[29]
ANDNOT 3.00  ; LS7 rotary table
ORLD
LD HR11.01  ; ROTALY TABLE UP/
ANDNOT 23.03  ; $?St$Bk?_#[30] / ALARM RESET / 堎$?St$Bk?_#[30]
ORLD
ANDLD
OUT HR11.01  ; ROTALY TABLE UP/

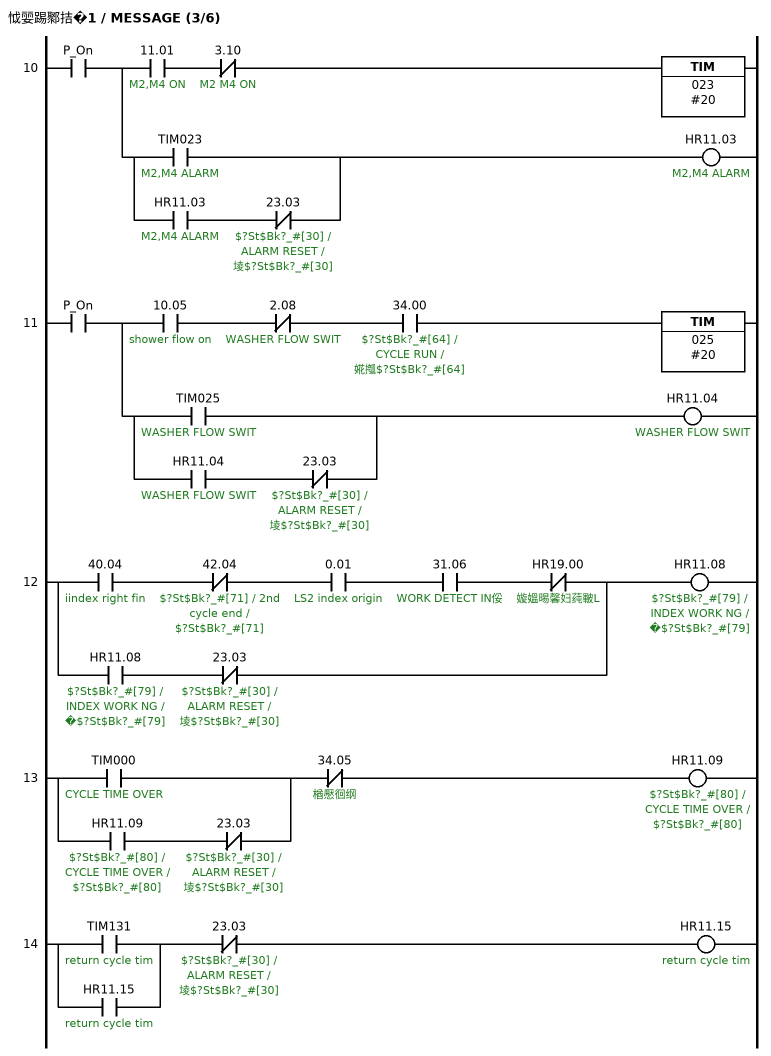
; rung 10
LD P_On
OUT TR0
AND 11.01  ; M2,M4 ON
ANDNOT 3.10  ; M2 M4 ON
TIM 023 #20
LD TR0
LD TIM023  ; M2,M4 ALARM
LD HR11.03  ; M2,M4 ALARM
ANDNOT 23.03  ; $?St$Bk?_#[30] / ALARM RESET / 堎$?St$Bk?_#[30]
ORLD
ANDLD
OUT HR11.03  ; M2,M4 ALARM
; rung 11
LD P_On
OUT TR0
AND 10.05  ; shower flow on
ANDNOT 2.08  ; WASHER FLOW SWIT
AND 34.00  ; $?St$Bk?_#[64] / CYCLE RUN / 婲摦$?St$Bk?_#[64]
TIM 025 #20
LD TR0
LD TIM025  ; WASHER FLOW SWIT
LD HR11.04  ; WASHER FLOW SWIT
ANDNOT 23.03  ; $?St$Bk?_#[30] / ALARM RESET / 堎$?St$Bk?_#[30]
ORLD
ANDLD
OUT HR11.04  ; WASHER FLOW SWIT
; rung 12
LD 40.04  ; iindex right fin
ANDNOT 42.04  ; $?St$Bk?_#[71] / 2nd cycle end / $?St$Bk?_#[71]
AND 0.01  ; LS2 index origin
AND 31.06  ; WORK DETECT IN俀
ANDNOT HR19.00  ; 嫙媼晹馨妇莼皸L
LD HR11.08  ; $?St$Bk?_#[79] / INDEX WORK NG / �$?St$Bk?_#[79]
ANDNOT 23.03  ; $?St$Bk?_#[30] / ALARM RESET / 堎$?St$Bk?_#[30]
ORLD
OUT HR11.08  ; $?St$Bk?_#[79] / INDEX WORK NG / �$?St$Bk?_#[79]
; rung 13
LD TIM000  ; CYCLE TIME OVER
LD HR11.09  ; $?St$Bk?_#[80] / CYCLE TIME OVER / $?St$Bk?_#[80]
ANDNOT 23.03  ; $?St$Bk?_#[30] / ALARM RESET / 堎$?St$Bk?_#[30]
ORLD
ANDNOT 34.05  ; 楢懕徊纲
OUT HR11.09  ; $?St$Bk?_#[80] / CYCLE TIME OVER / $?St$Bk?_#[80]
; rung 14
LD TIM131  ; return cycle tim
OR HR11.15  ; return cycle tim
ANDNOT 23.03  ; $?St$Bk?_#[30] / ALARM RESET / 堎$?St$Bk?_#[30]
OUT HR11.15  ; return cycle tim

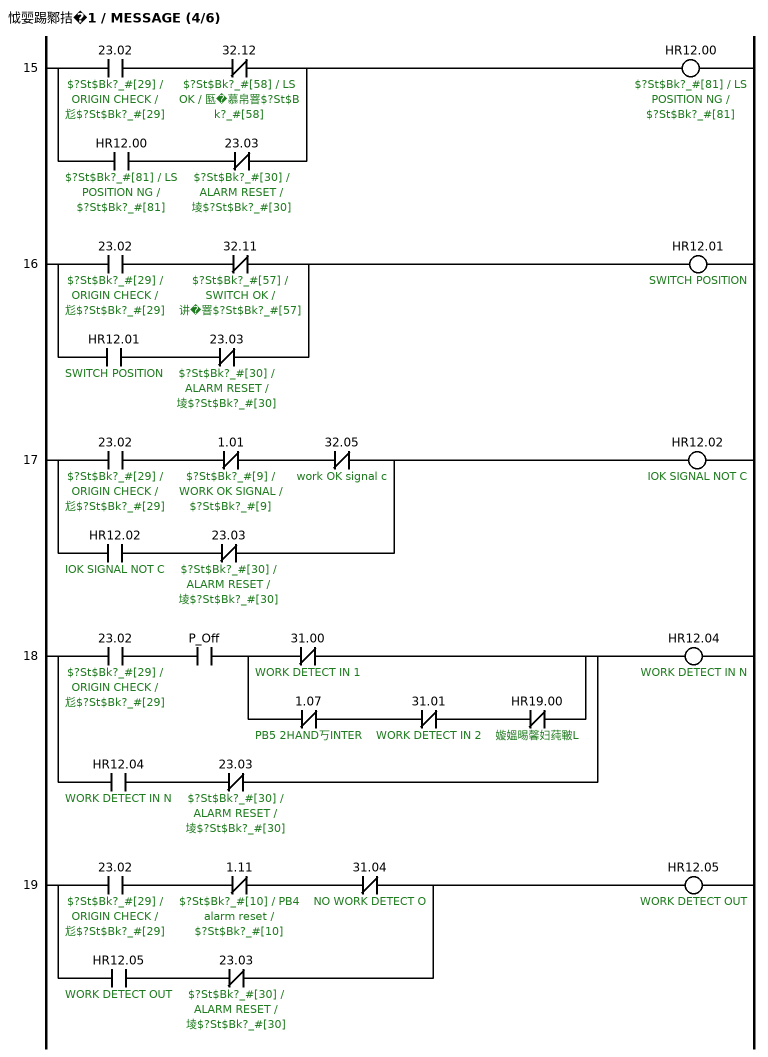
; rung 15
LD 23.02  ; $?St$Bk?_#[29] / ORIGIN CHECK / 尨$?St$Bk?_#[29]
ANDNOT 32.12  ; $?St$Bk?_#[58] / LS OK / 匦�慕帛罯$?St$Bk?_#[58]
LD HR12.00  ; $?St$Bk?_#[81] / LS POSITION NG / $?St$Bk?_#[81]
ANDNOT 23.03  ; $?St$Bk?_#[30] / ALARM RESET / 堎$?St$Bk?_#[30]
ORLD
OUT HR12.00  ; $?St$Bk?_#[81] / LS POSITION NG / $?St$Bk?_#[81]
; rung 16
LD 23.02  ; $?St$Bk?_#[29] / ORIGIN CHECK / 尨$?St$Bk?_#[29]
ANDNOT 32.11  ; $?St$Bk?_#[57] / SWITCH OK / 讲�罯$?St$Bk?_#[57]
LD HR12.01  ; SWITCH POSITION
ANDNOT 23.03  ; $?St$Bk?_#[30] / ALARM RESET / 堎$?St$Bk?_#[30]
ORLD
OUT HR12.01  ; SWITCH POSITION
; rung 17
LD 23.02  ; $?St$Bk?_#[29] / ORIGIN CHECK / 尨$?St$Bk?_#[29]
ANDNOT 1.01  ; $?St$Bk?_#[9] / WORK OK SIGNAL / $?St$Bk?_#[9]
ANDNOT 32.05  ; work OK signal c
LD HR12.02  ; IOK SIGNAL NOT C
ANDNOT 23.03  ; $?St$Bk?_#[30] / ALARM RESET / 堎$?St$Bk?_#[30]
ORLD
OUT HR12.02  ; IOK SIGNAL NOT C
; rung 18
LD 23.02  ; $?St$Bk?_#[29] / ORIGIN CHECK / 尨$?St$Bk?_#[29]
AND P_Off
LDNOT 31.00  ; WORK DETECT IN 1
LDNOT 1.07  ; PB5 2HAND丂INTER
ANDNOT 31.01  ; WORK DETECT IN 2
ANDNOT HR19.00  ; 嫙媼晹馨妇莼皸L
ORLD
ANDLD
LD HR12.04  ; WORK DETECT IN N
ANDNOT 23.03  ; $?St$Bk?_#[30] / ALARM RESET / 堎$?St$Bk?_#[30]
ORLD
OUT HR12.04  ; WORK DETECT IN N
; rung 19
LD 23.02  ; $?St$Bk?_#[29] / ORIGIN CHECK / 尨$?St$Bk?_#[29]
ANDNOT 1.11  ; $?St$Bk?_#[10] / PB4 alarm reset / $?St$Bk?_#[10]
ANDNOT 31.04  ; NO WORK DETECT O
LD HR12.05  ; WORK DETECT OUT
ANDNOT 23.03  ; $?St$Bk?_#[30] / ALARM RESET / 堎$?St$Bk?_#[30]
ORLD
OUT HR12.05  ; WORK DETECT OUT

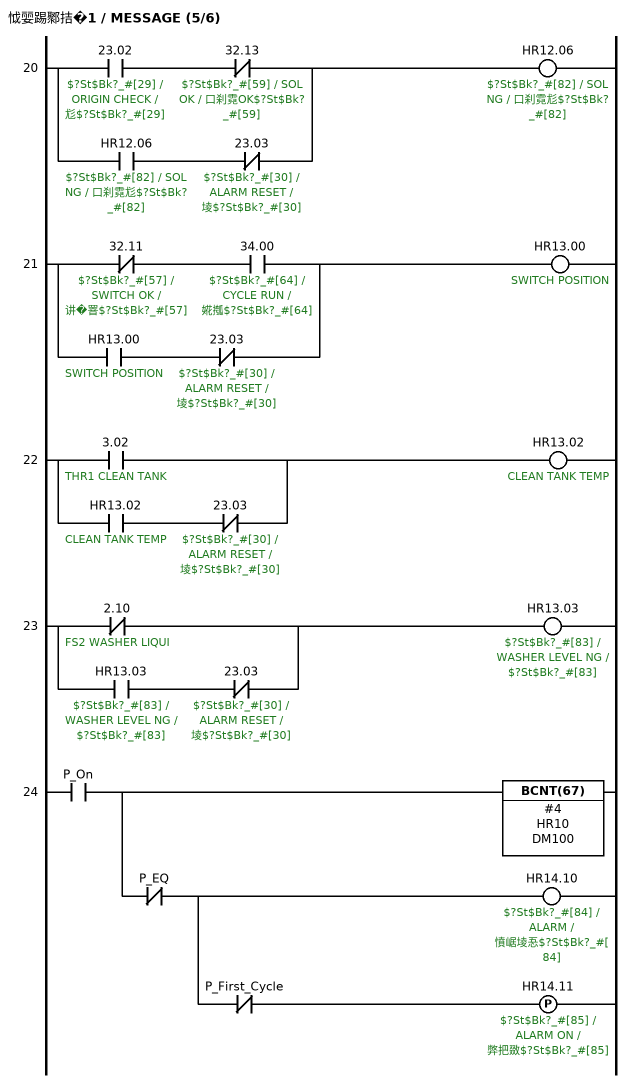
; rung 20
LD 23.02  ; $?St$Bk?_#[29] / ORIGIN CHECK / 尨$?St$Bk?_#[29]
ANDNOT 32.13  ; $?St$Bk?_#[59] / SOL OK / 口刹霓OK$?St$Bk?_#[59]
LD HR12.06  ; $?St$Bk?_#[82] / SOL NG / 口刹霓尨$?St$Bk?_#[82]
ANDNOT 23.03  ; $?St$Bk?_#[30] / ALARM RESET / 堎$?St$Bk?_#[30]
ORLD
OUT HR12.06  ; $?St$Bk?_#[82] / SOL NG / 口刹霓尨$?St$Bk?_#[82]
; rung 21
LDNOT 32.11  ; $?St$Bk?_#[57] / SWITCH OK / 讲�罯$?St$Bk?_#[57]
AND 34.00  ; $?St$Bk?_#[64] / CYCLE RUN / 婲摦$?St$Bk?_#[64]
LD HR13.00  ; SWITCH POSITION
ANDNOT 23.03  ; $?St$Bk?_#[30] / ALARM RESET / 堎$?St$Bk?_#[30]
ORLD
OUT HR13.00  ; SWITCH POSITION
; rung 22
LD 3.02  ; THR1 CLEAN TANK
LD HR13.02  ; CLEAN TANK TEMP
ANDNOT 23.03  ; $?St$Bk?_#[30] / ALARM RESET / 堎$?St$Bk?_#[30]
ORLD
OUT HR13.02  ; CLEAN TANK TEMP
; rung 23
LDNOT 2.10  ; FS2 WASHER LIQUI
LD HR13.03  ; $?St$Bk?_#[83] / WASHER LEVEL NG / $?St$Bk?_#[83]
ANDNOT 23.03  ; $?St$Bk?_#[30] / ALARM RESET / 堎$?St$Bk?_#[30]
ORLD
OUT HR13.03  ; $?St$Bk?_#[83] / WASHER LEVEL NG / $?St$Bk?_#[83]
; rung 24
LD P_On
BCNT(67) #4 HR10 DM100
ANDNOT P_EQ
OUT HR14.10  ; $?St$Bk?_#[84] / ALARM / 憤崌堎忢$?St$Bk?_#[84]
ANDNOT P_First_Cycle
DIFU(13) HR14.11  ; $?St$Bk?_#[85] / ALARM ON / 弊把敪$?St$Bk?_#[85]

